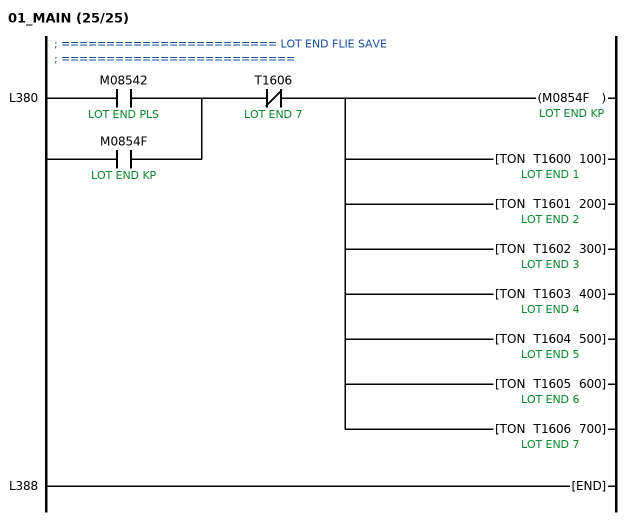
[picture p24: 01_MAIN rungs L380-L388]
// ======================== LOT END FLIE SAVE ==========================
; L380
LOAD      M08542	// LOT END PLS
OR        M0854F	// LOT END KP
AND NOT   T1606	// LOT END 7
OUT       M0854F	// LOT END KP
TON       T1600 100	// LOT END 1
TON       T1601 200	// LOT END 2
TON       T1602 300	// LOT END 3
TON       T1603 400	// LOT END 4
TON       T1604 500	// LOT END 5
TON       T1605 600	// LOT END 6
TON       T1606 700	// LOT END 7
; L388
END

PROGRAM 02_AUTO_RUN (task: ½ºÄµ ÇÁ·Î±×·¥)

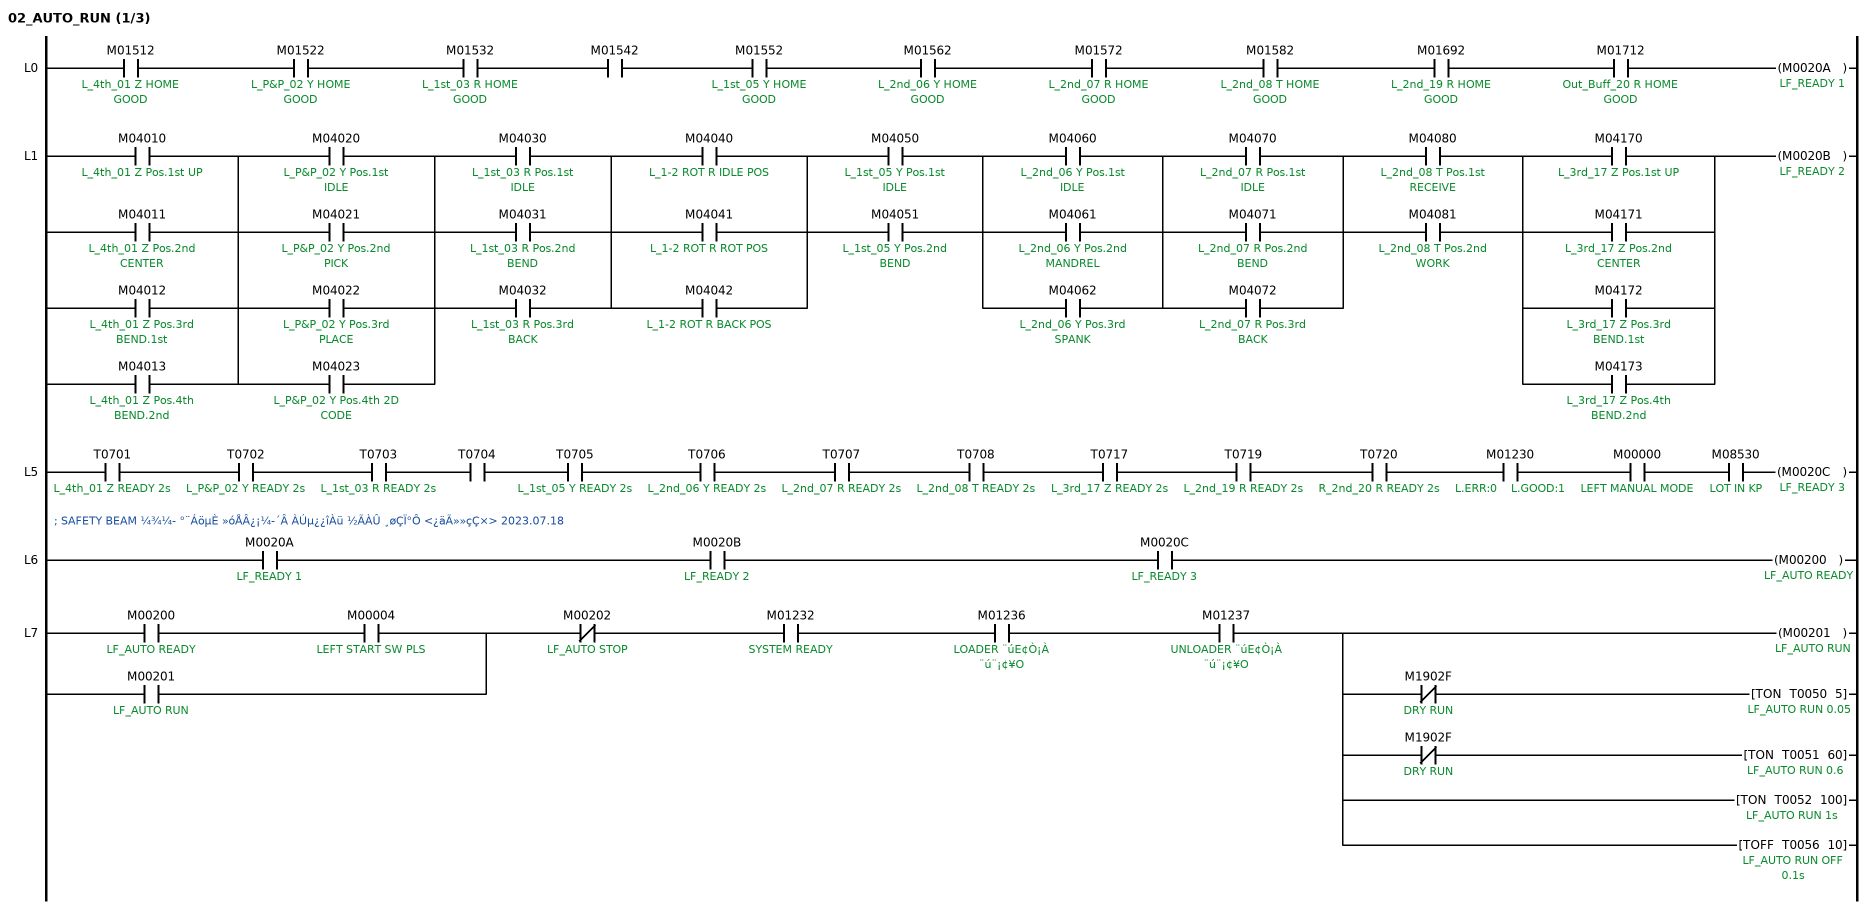
; L0
LOAD      M01512	// L_4th_01 Z HOME GOOD
AND       M01522	// L_P&P_02 Y HOME GOOD
AND       M01532	// L_1st_03 R HOME GOOD
AND       M01542
AND       M01552	// L_1st_05 Y HOME GOOD
AND       M01562	// L_2nd_06 Y HOME GOOD
AND       M01572	// L_2nd_07 R HOME GOOD
AND       M01582	// L_2nd_08 T HOME GOOD
AND       M01692	// L_2nd_19 R HOME GOOD
AND       M01712	// Out_Buff_20 R HOME GOOD
OUT       M0020A	// LF_READY 1
; L1
LOAD      M04010	// L_4th_01 Z Pos.1st UP
OR        M04011	// L_4th_01 Z Pos.2nd CENTER
OR        M04012	// L_4th_01 Z Pos.3rd BEND.1st
OR        M04013	// L_4th_01 Z Pos.4th BEND.2nd
LOAD      M04020	// L_P&P_02 Y Pos.1st IDLE
OR        M04021	// L_P&P_02 Y Pos.2nd PICK
OR        M04022	// L_P&P_02 Y Pos.3rd PLACE
OR        M04023	// L_P&P_02 Y Pos.4th 2D CODE
AND LOAD
LOAD      M04030	// L_1st_03 R Pos.1st IDLE
OR        M04031	// L_1st_03 R Pos.2nd BEND
OR        M04032	// L_1st_03 R Pos.3rd BACK
AND LOAD
LOAD      M04040	// L_1-2 ROT R IDLE POS
OR        M04041	// L_1-2 ROT R ROT POS
OR        M04042	// L_1-2 ROT R BACK POS
AND LOAD
LOAD      M04050	// L_1st_05 Y Pos.1st IDLE
OR        M04051	// L_1st_05 Y Pos.2nd BEND
AND LOAD
LOAD      M04060	// L_2nd_06 Y Pos.1st IDLE
OR        M04061	// L_2nd_06 Y Pos.2nd MANDREL
OR        M04062	// L_2nd_06 Y Pos.3rd SPANK
AND LOAD
LOAD      M04070	// L_2nd_07 R Pos.1st IDLE
OR        M04071	// L_2nd_07 R Pos.2nd BEND
OR        M04072	// L_2nd_07 R Pos.3rd BACK
AND LOAD
LOAD      M04080	// L_2nd_08 T Pos.1st RECEIVE
OR        M04081	// L_2nd_08 T Pos.2nd WORK
AND LOAD
LOAD      M04170	// L_3rd_17 Z Pos.1st UP
OR        M04171	// L_3rd_17 Z Pos.2nd CENTER
OR        M04172	// L_3rd_17 Z Pos.3rd BEND.1st
OR        M04173	// L_3rd_17 Z Pos.4th BEND.2nd
AND LOAD
OUT       M0020B	// LF_READY 2
; L5
LOAD      T0701	// L_4th_01 Z READY 2s
AND       T0702	// L_P&P_02 Y READY 2s
AND       T0703	// L_1st_03 R READY 2s
AND       T0704
AND       T0705	// L_1st_05 Y READY 2s
AND       T0706	// L_2nd_06 Y READY 2s
AND       T0707	// L_2nd_07 R READY 2s
AND       T0708	// L_2nd_08 T READY 2s
AND       T0717	// L_3rd_17 Z READY 2s
AND       T0719	// L_2nd_19 R READY 2s
AND       T0720	// R_2nd_20 R READY 2s
AND       M01230	// L.ERR:0    L.GOOD:1
AND       M00000	// LEFT MANUAL MODE
AND       M08530	// LOT IN KP
OUT       M0020C	// LF_READY 3
; L6
LOAD      M0020A	// LF_READY 1
AND       M0020B	// LF_READY 2
AND       M0020C	// LF_READY 3
OUT       M00200	// LF_AUTO READY
// output comment: SAFETY BEAM ¼¾¼­ °¨ÁöµÈ »óÅÂ¿¡¼­´Â ÀÚµ¿¿îÀü ½ÃÀÛ ¸øÇÏ°Ô <¿äÃ»»çÇ×> 2023.07.18
; L7
LOAD      M00200	// LF_AUTO READY
AND       M00004	// LEFT START SW PLS
OR        M00201	// LF_AUTO RUN
AND NOT   M00202	// LF_AUTO STOP
AND       M01232	// SYSTEM READY
AND       M01236	// LOADER ¨úE¢Ò¡À ¨ú¨¡¢¥O
AND       M01237	// UNLOADER ¨úE¢Ò¡À ¨ú¨¡¢¥O
OUT       M00201	// LF_AUTO RUN
MPUSH
AND NOT   M1902F	// DRY RUN
TON       T0050 5	// LF_AUTO RUN 0.05
MLOAD
AND NOT   M1902F	// DRY RUN
TON       T0051 60	// LF_AUTO RUN 0.6
MPOP
TON       T0052 100	// LF_AUTO RUN 1s
TOFF      T0056 10	// LF_AUTO RUN OFF 0.1s

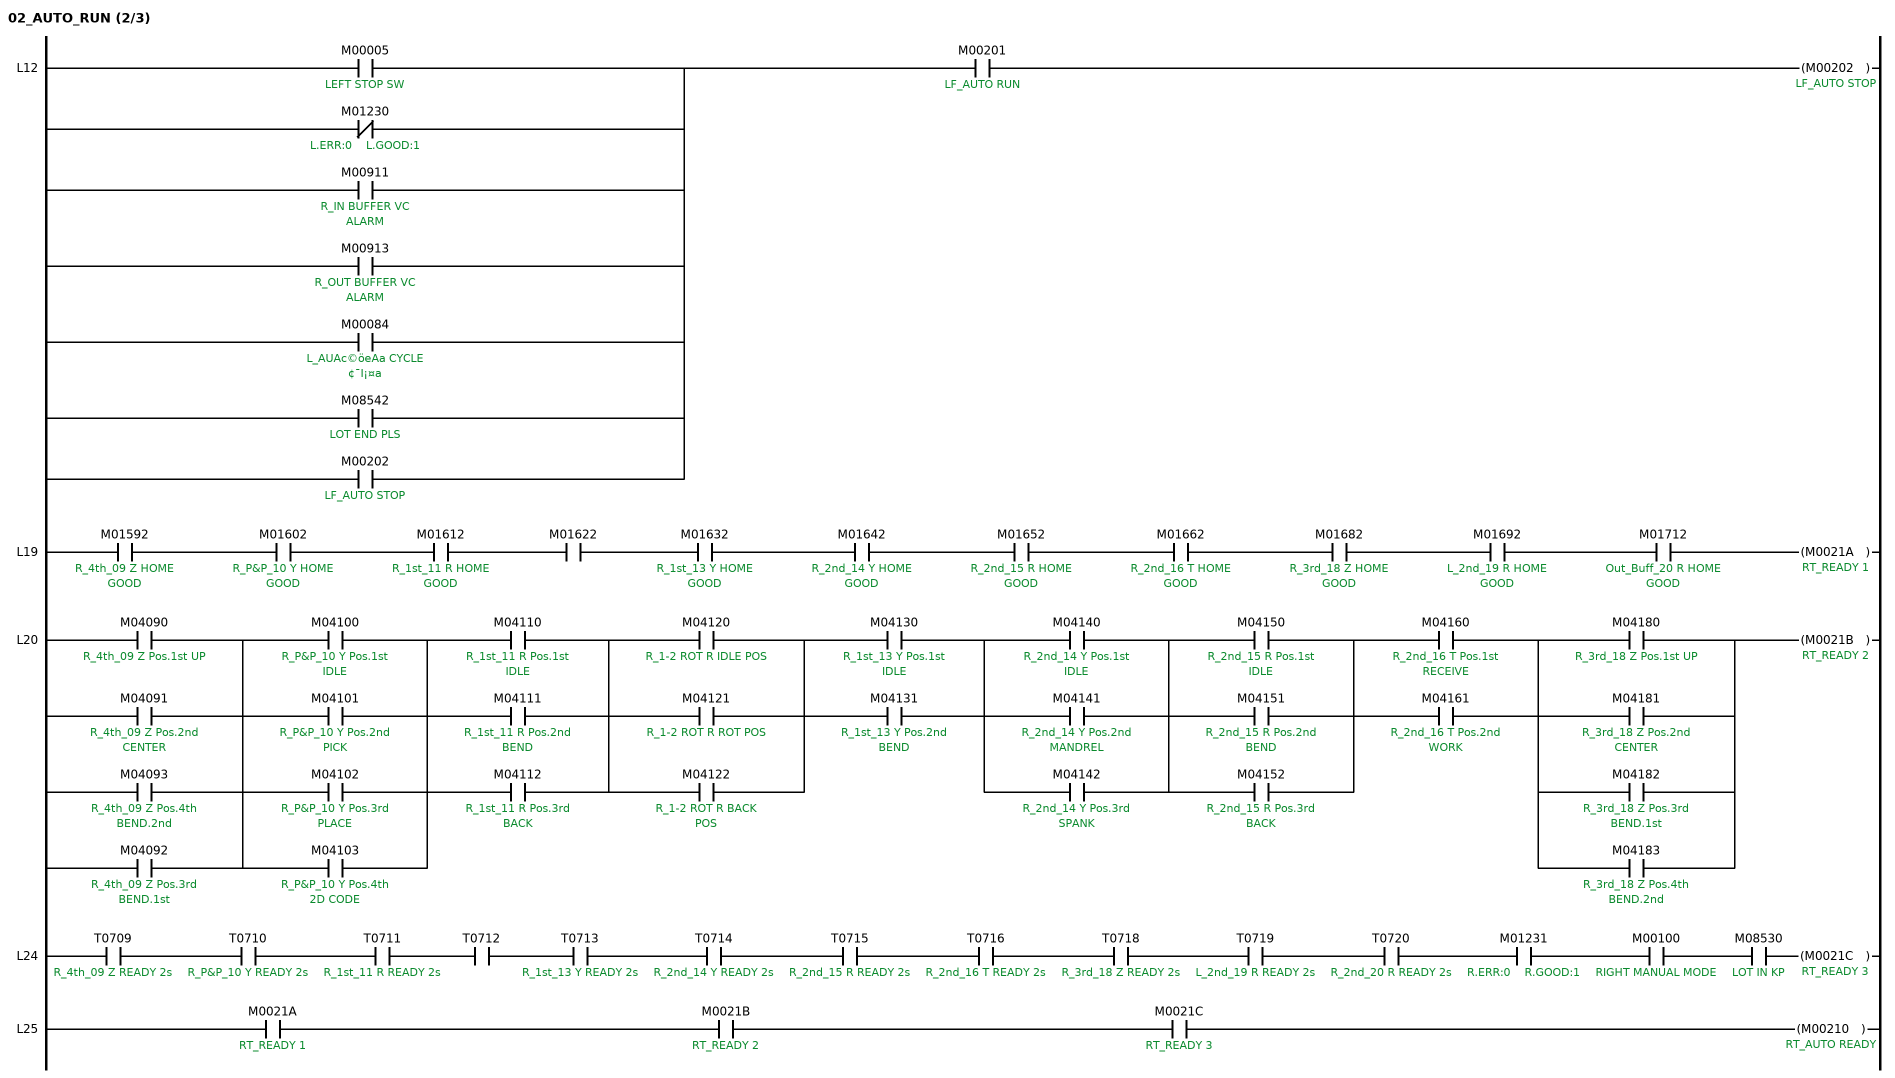
; L12
LOAD      M00005	// LEFT STOP SW
OR NOT    M01230	// L.ERR:0    L.GOOD:1
OR        M00911	// R_IN BUFFER VC ALARM
OR        M00913	// R_OUT BUFFER VC ALARM
OR        M00084	// L_AUAc©öeAa CYCLE ¢¯I¡¤a
OR        M08542	// LOT END PLS
OR        M00202	// LF_AUTO STOP
AND       M00201	// LF_AUTO RUN
OUT       M00202	// LF_AUTO STOP
; L19
LOAD      M01592	// R_4th_09 Z HOME GOOD
AND       M01602	// R_P&P_10 Y HOME GOOD
AND       M01612	// R_1st_11 R HOME GOOD
AND       M01622
AND       M01632	// R_1st_13 Y HOME GOOD
AND       M01642	// R_2nd_14 Y HOME GOOD
AND       M01652	// R_2nd_15 R HOME GOOD
AND       M01662	// R_2nd_16 T HOME GOOD
AND       M01682	// R_3rd_18 Z HOME GOOD
AND       M01692	// L_2nd_19 R HOME GOOD
AND       M01712	// Out_Buff_20 R HOME GOOD
OUT       M0021A	// RT_READY 1
; L20
LOAD      M04090	// R_4th_09 Z Pos.1st UP
OR        M04091	// R_4th_09 Z Pos.2nd CENTER
OR        M04093	// R_4th_09 Z Pos.4th BEND.2nd
OR        M04092	// R_4th_09 Z Pos.3rd BEND.1st
LOAD      M04100	// R_P&P_10 Y Pos.1st IDLE
OR        M04101	// R_P&P_10 Y Pos.2nd PICK
OR        M04102	// R_P&P_10 Y Pos.3rd PLACE
OR        M04103	// R_P&P_10 Y Pos.4th 2D CODE
AND LOAD
LOAD      M04110	// R_1st_11 R Pos.1st IDLE
OR        M04111	// R_1st_11 R Pos.2nd BEND
OR        M04112	// R_1st_11 R Pos.3rd BACK
AND LOAD
LOAD      M04120	// R_1-2 ROT R IDLE POS
OR        M04121	// R_1-2 ROT R ROT POS
OR        M04122	// R_1-2 ROT R BACK POS
AND LOAD
LOAD      M04130	// R_1st_13 Y Pos.1st IDLE
OR        M04131	// R_1st_13 Y Pos.2nd BEND
AND LOAD
LOAD      M04140	// R_2nd_14 Y Pos.1st IDLE
OR        M04141	// R_2nd_14 Y Pos.2nd MANDREL
OR        M04142	// R_2nd_14 Y Pos.3rd SPANK
AND LOAD
LOAD      M04150	// R_2nd_15 R Pos.1st IDLE
OR        M04151	// R_2nd_15 R Pos.2nd BEND
OR        M04152	// R_2nd_15 R Pos.3rd BACK
AND LOAD
LOAD      M04160	// R_2nd_16 T Pos.1st RECEIVE
OR        M04161	// R_2nd_16 T Pos.2nd WORK
AND LOAD
LOAD      M04180	// R_3rd_18 Z Pos.1st UP
OR        M04181	// R_3rd_18 Z Pos.2nd CENTER
OR        M04182	// R_3rd_18 Z Pos.3rd BEND.1st
OR        M04183	// R_3rd_18 Z Pos.4th BEND.2nd
AND LOAD
OUT       M0021B	// RT_READY 2
; L24
LOAD      T0709	// R_4th_09 Z READY 2s
AND       T0710	// R_P&P_10 Y READY 2s
AND       T0711	// R_1st_11 R READY 2s
AND       T0712
AND       T0713	// R_1st_13 Y READY 2s
AND       T0714	// R_2nd_14 Y READY 2s
AND       T0715	// R_2nd_15 R READY 2s
AND       T0716	// R_2nd_16 T READY 2s
AND       T0718	// R_3rd_18 Z READY 2s
AND       T0719	// L_2nd_19 R READY 2s
AND       T0720	// R_2nd_20 R READY 2s
AND       M01231	// R.ERR:0    R.GOOD:1
AND       M00100	// RIGHT MANUAL MODE
AND       M08530	// LOT IN KP
OUT       M0021C	// RT_READY 3
; L25
LOAD      M0021A	// RT_READY 1
AND       M0021B	// RT_READY 2
AND       M0021C	// RT_READY 3
OUT       M00210	// RT_AUTO READY

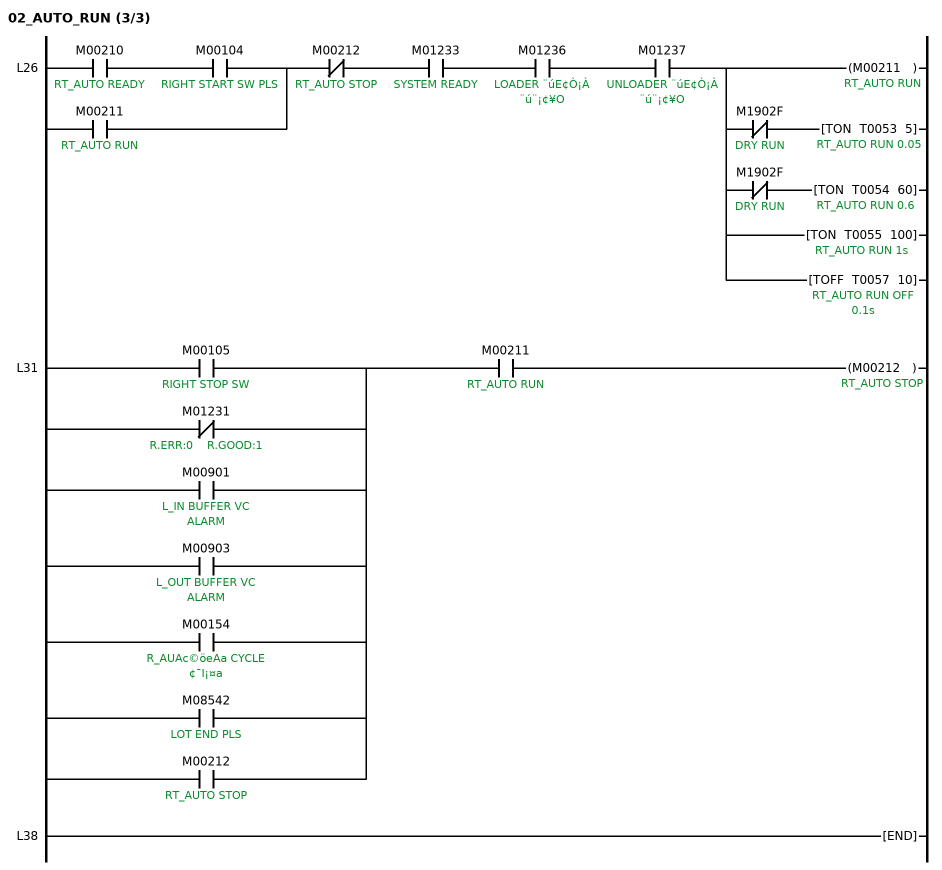
; L26
LOAD      M00210	// RT_AUTO READY
AND       M00104	// RIGHT START SW PLS
OR        M00211	// RT_AUTO RUN
AND NOT   M00212	// RT_AUTO STOP
AND       M01233	// SYSTEM READY
AND       M01236	// LOADER ¨úE¢Ò¡À ¨ú¨¡¢¥O
AND       M01237	// UNLOADER ¨úE¢Ò¡À ¨ú¨¡¢¥O
OUT       M00211	// RT_AUTO RUN
MPUSH
AND NOT   M1902F	// DRY RUN
TON       T0053 5	// RT_AUTO RUN 0.05
MLOAD
AND NOT   M1902F	// DRY RUN
TON       T0054 60	// RT_AUTO RUN 0.6
MPOP
TON       T0055 100	// RT_AUTO RUN 1s
TOFF      T0057 10	// RT_AUTO RUN OFF 0.1s
; L31
LOAD      M00105	// RIGHT STOP SW
OR NOT    M01231	// R.ERR:0    R.GOOD:1
OR        M00901	// L_IN BUFFER VC ALARM
OR        M00903	// L_OUT BUFFER VC ALARM
OR        M00154	// R_AUAc©öeAa CYCLE ¢¯I¡¤a
OR        M08542	// LOT END PLS
OR        M00212	// RT_AUTO STOP
AND       M00211	// RT_AUTO RUN
OUT       M00212	// RT_AUTO STOP
; L38
END

PROGRAM 03_COUNT (task: ½ºÄµ ÇÁ·Î±×·¥)

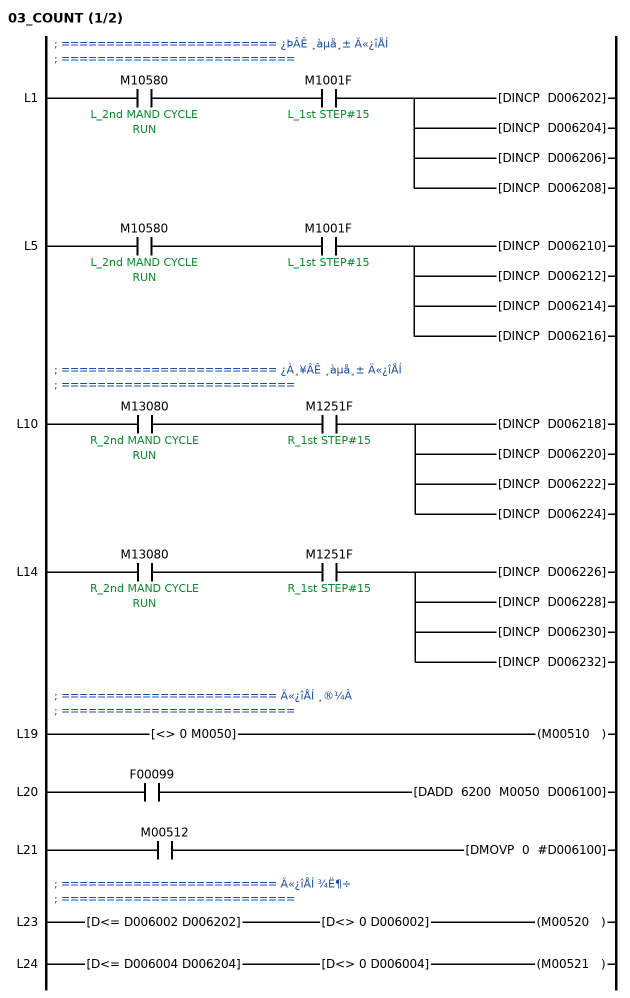
// ======================== ¿ÞÂÊ ¸àµå¸± Ä«¿îÅÍ ==========================
; L1
LOAD      M10580	// L_2nd MAND CYCLE RUN
AND       M1001F	// L_1st STEP#15
DINCP     D006202
DINCP     D006204
DINCP     D006206
DINCP     D006208
; L5
LOAD      M10580	// L_2nd MAND CYCLE RUN
AND       M1001F	// L_1st STEP#15
DINCP     D006210
DINCP     D006212
DINCP     D006214
DINCP     D006216
// ======================== ¿À¸¥ÂÊ ¸àµå¸± Ä«¿îÅÍ ==========================
; L10
LOAD      M13080	// R_2nd MAND CYCLE RUN
AND       M1251F	// R_1st STEP#15
DINCP     D006218
DINCP     D006220
DINCP     D006222
DINCP     D006224
; L14
LOAD      M13080	// R_2nd MAND CYCLE RUN
AND       M1251F	// R_1st STEP#15
DINCP     D006226
DINCP     D006228
DINCP     D006230
DINCP     D006232
// ======================== Ä«¿îÅÍ ¸®¼Â ==========================
; L19
LOAD<>    0 M0050
OUT       M00510
; L20
LOAD      F00099
DADD      6200 M0050 D006100
; L21
LOAD      M00512
DMOVP     0 #D006100
// ======================== Ä«¿îÅÍ ¾Ë¶÷ ==========================
; L23
LOADD<=   D006002 D006202
ANDD<>    0 D006002
OUT       M00520
; L24
LOADD<=   D006004 D006204
ANDD<>    0 D006004
OUT       M00521

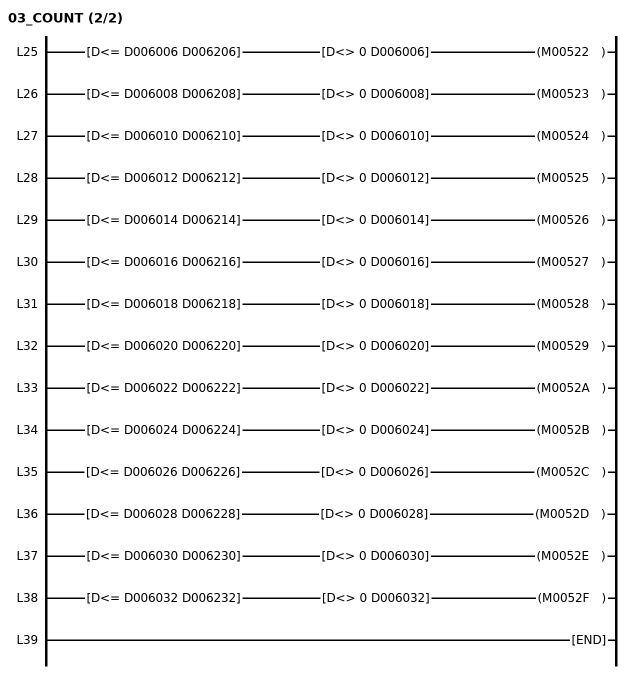
; L25
LOADD<=   D006006 D006206
ANDD<>    0 D006006
OUT       M00522
; L26
LOADD<=   D006008 D006208
ANDD<>    0 D006008
OUT       M00523
; L27
LOADD<=   D006010 D006210
ANDD<>    0 D006010
OUT       M00524
; L28
LOADD<=   D006012 D006212
ANDD<>    0 D006012
OUT       M00525
; L29
LOADD<=   D006014 D006214
ANDD<>    0 D006014
OUT       M00526
; L30
LOADD<=   D006016 D006216
ANDD<>    0 D006016
OUT       M00527
; L31
LOADD<=   D006018 D006218
ANDD<>    0 D006018
OUT       M00528
; L32
LOADD<=   D006020 D006220
ANDD<>    0 D006020
OUT       M00529
; L33
LOADD<=   D006022 D006222
ANDD<>    0 D006022
OUT       M0052A
; L34
LOADD<=   D006024 D006224
ANDD<>    0 D006024
OUT       M0052B
; L35
LOADD<=   D006026 D006226
ANDD<>    0 D006026
OUT       M0052C
; L36
LOADD<=   D006028 D006228
ANDD<>    0 D006028
OUT       M0052D
; L37
LOADD<=   D006030 D006230
ANDD<>    0 D006030
OUT       M0052E
; L38
LOADD<=   D006032 D006232
ANDD<>    0 D006032
OUT       M0052F
; L39
END

PROGRAM 04_VACUUM_FLOW (task: ½ºÄµ ÇÁ·Î±×·¥)

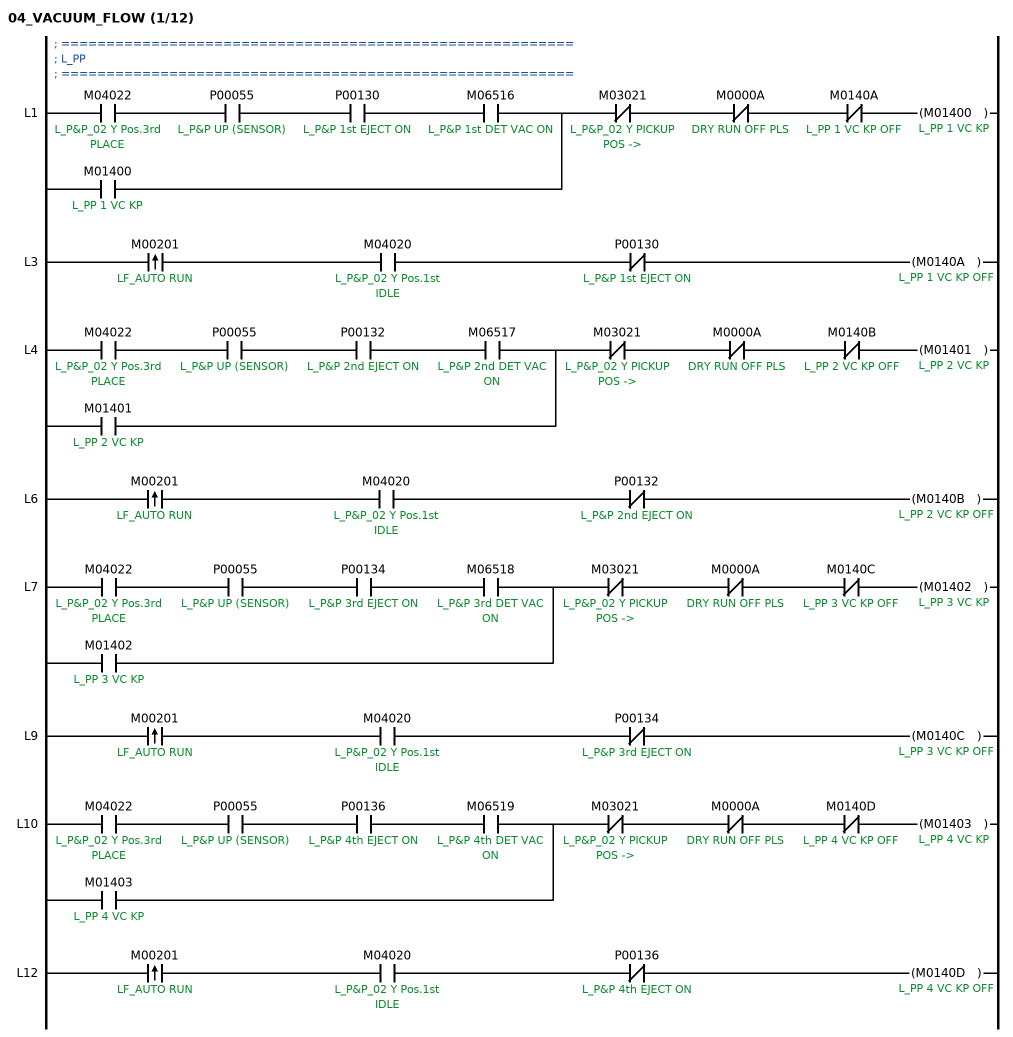
// =========================================================
// 
//       L_PP
// 
// =========================================================
; L1
LOAD      M04022	// L_P&P_02 Y Pos.3rd PLACE
AND       P00055	// L_P&P UP (SENSOR)
AND       P00130	// L_P&P 1st EJECT ON
AND       M06516	// L_P&P 1st DET VAC ON
OR        M01400	// L_PP 1 VC KP
AND NOT   M03021	// L_P&P_02 Y PICKUP POS ->
AND NOT   M0000A	// DRY RUN OFF PLS
AND NOT   M0140A	// L_PP 1 VC KP OFF
OUT       M01400	// L_PP 1 VC KP
; L3
LOADP     M00201	// LF_AUTO RUN
AND       M04020	// L_P&P_02 Y Pos.1st IDLE
AND NOT   P00130	// L_P&P 1st EJECT ON
OUT       M0140A	// L_PP 1 VC KP OFF
; L4
LOAD      M04022	// L_P&P_02 Y Pos.3rd PLACE
AND       P00055	// L_P&P UP (SENSOR)
AND       P00132	// L_P&P 2nd EJECT ON
AND       M06517	// L_P&P 2nd DET VAC ON
OR        M01401	// L_PP 2 VC KP
AND NOT   M03021	// L_P&P_02 Y PICKUP POS ->
AND NOT   M0000A	// DRY RUN OFF PLS
AND NOT   M0140B	// L_PP 2 VC KP OFF
OUT       M01401	// L_PP 2 VC KP
; L6
LOADP     M00201	// LF_AUTO RUN
AND       M04020	// L_P&P_02 Y Pos.1st IDLE
AND NOT   P00132	// L_P&P 2nd EJECT ON
OUT       M0140B	// L_PP 2 VC KP OFF
; L7
LOAD      M04022	// L_P&P_02 Y Pos.3rd PLACE
AND       P00055	// L_P&P UP (SENSOR)
AND       P00134	// L_P&P 3rd EJECT ON
AND       M06518	// L_P&P 3rd DET VAC ON
OR        M01402	// L_PP 3 VC KP
AND NOT   M03021	// L_P&P_02 Y PICKUP POS ->
AND NOT   M0000A	// DRY RUN OFF PLS
AND NOT   M0140C	// L_PP 3 VC KP OFF
OUT       M01402	// L_PP 3 VC KP
; L9
LOADP     M00201	// LF_AUTO RUN
AND       M04020	// L_P&P_02 Y Pos.1st IDLE
AND NOT   P00134	// L_P&P 3rd EJECT ON
OUT       M0140C	// L_PP 3 VC KP OFF
; L10
LOAD      M04022	// L_P&P_02 Y Pos.3rd PLACE
AND       P00055	// L_P&P UP (SENSOR)
AND       P00136	// L_P&P 4th EJECT ON
AND       M06519	// L_P&P 4th DET VAC ON
OR        M01403	// L_PP 4 VC KP
AND NOT   M03021	// L_P&P_02 Y PICKUP POS ->
AND NOT   M0000A	// DRY RUN OFF PLS
AND NOT   M0140D	// L_PP 4 VC KP OFF
OUT       M01403	// L_PP 4 VC KP
; L12
LOADP     M00201	// LF_AUTO RUN
AND       M04020	// L_P&P_02 Y Pos.1st IDLE
AND NOT   P00136	// L_P&P 4th EJECT ON
OUT       M0140D	// L_PP 4 VC KP OFF

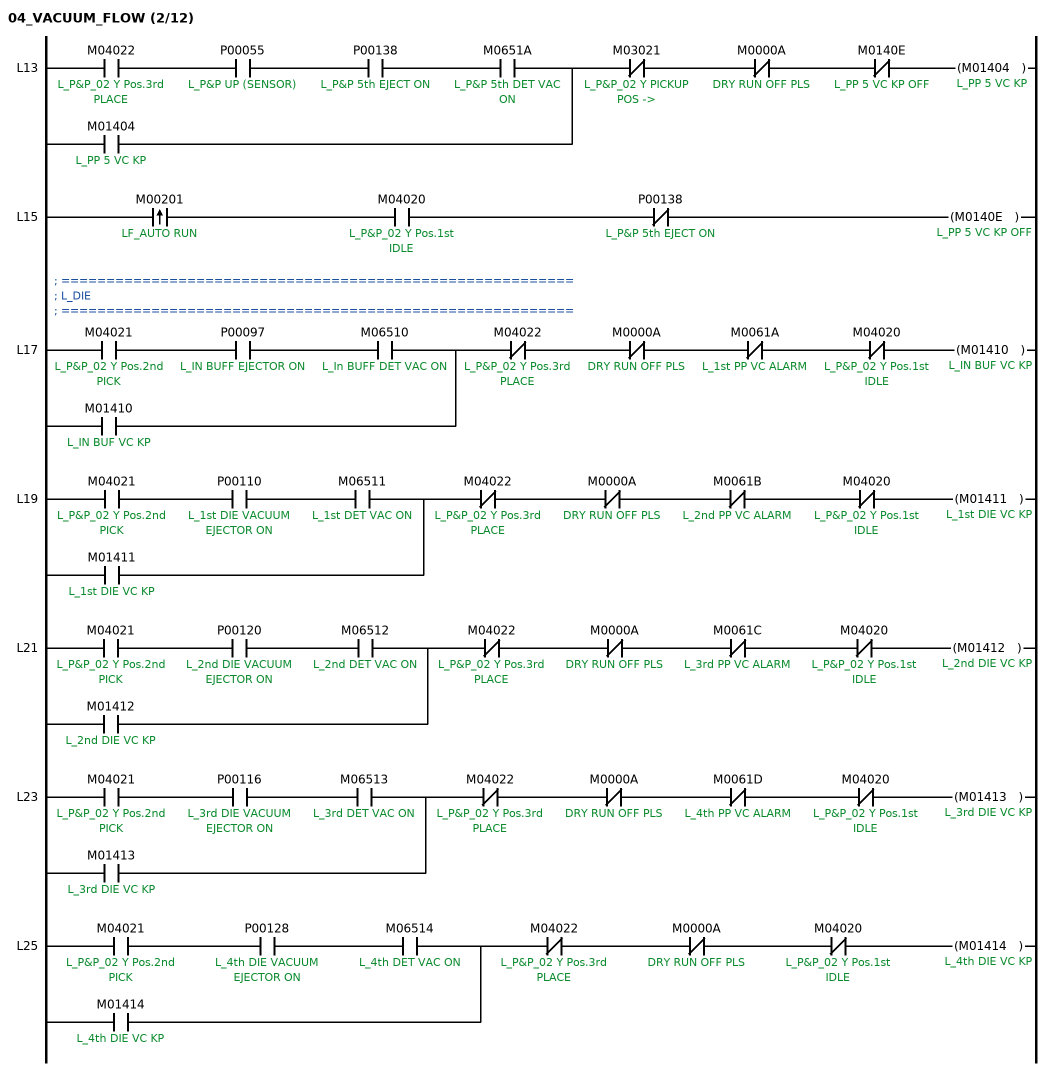
; L13
LOAD      M04022	// L_P&P_02 Y Pos.3rd PLACE
AND       P00055	// L_P&P UP (SENSOR)
AND       P00138	// L_P&P 5th EJECT ON
AND       M0651A	// L_P&P 5th DET VAC ON
OR        M01404	// L_PP 5 VC KP
AND NOT   M03021	// L_P&P_02 Y PICKUP POS ->
AND NOT   M0000A	// DRY RUN OFF PLS
AND NOT   M0140E	// L_PP 5 VC KP OFF
OUT       M01404	// L_PP 5 VC KP
; L15
LOADP     M00201	// LF_AUTO RUN
AND       M04020	// L_P&P_02 Y Pos.1st IDLE
AND NOT   P00138	// L_P&P 5th EJECT ON
OUT       M0140E	// L_PP 5 VC KP OFF
// =========================================================
// 
//       L_DIE
// 
// =========================================================
; L17
LOAD      M04021	// L_P&P_02 Y Pos.2nd PICK
AND       P00097	// L_IN BUFF EJECTOR ON
AND       M06510	// L_In BUFF DET VAC ON
OR        M01410	// L_IN BUF VC KP
AND NOT   M04022	// L_P&P_02 Y Pos.3rd PLACE
AND NOT   M0000A	// DRY RUN OFF PLS
AND NOT   M0061A	// L_1st PP VC ALARM
AND NOT   M04020	// L_P&P_02 Y Pos.1st IDLE
OUT       M01410	// L_IN BUF VC KP
; L19
LOAD      M04021	// L_P&P_02 Y Pos.2nd PICK
AND       P00110	// L_1st DIE VACUUM EJECTOR ON
AND       M06511	// L_1st DET VAC ON
OR        M01411	// L_1st DIE VC KP
AND NOT   M04022	// L_P&P_02 Y Pos.3rd PLACE
AND NOT   M0000A	// DRY RUN OFF PLS
AND NOT   M0061B	// L_2nd PP VC ALARM
AND NOT   M04020	// L_P&P_02 Y Pos.1st IDLE
OUT       M01411	// L_1st DIE VC KP
; L21
LOAD      M04021	// L_P&P_02 Y Pos.2nd PICK
AND       P00120	// L_2nd DIE VACUUM EJECTOR ON
AND       M06512	// L_2nd DET VAC ON
OR        M01412	// L_2nd DIE VC KP
AND NOT   M04022	// L_P&P_02 Y Pos.3rd PLACE
AND NOT   M0000A	// DRY RUN OFF PLS
AND NOT   M0061C	// L_3rd PP VC ALARM
AND NOT   M04020	// L_P&P_02 Y Pos.1st IDLE
OUT       M01412	// L_2nd DIE VC KP
; L23
LOAD      M04021	// L_P&P_02 Y Pos.2nd PICK
AND       P00116	// L_3rd DIE VACUUM EJECTOR ON
AND       M06513	// L_3rd DET VAC ON
OR        M01413	// L_3rd DIE VC KP
AND NOT   M04022	// L_P&P_02 Y Pos.3rd PLACE
AND NOT   M0000A	// DRY RUN OFF PLS
AND NOT   M0061D	// L_4th PP VC ALARM
AND NOT   M04020	// L_P&P_02 Y Pos.1st IDLE
OUT       M01413	// L_3rd DIE VC KP
; L25
LOAD      M04021	// L_P&P_02 Y Pos.2nd PICK
AND       P00128	// L_4th DIE VACUUM EJECTOR ON
AND       M06514	// L_4th DET VAC ON
OR        M01414	// L_4th DIE VC KP
AND NOT   M04022	// L_P&P_02 Y Pos.3rd PLACE
AND NOT   M0000A	// DRY RUN OFF PLS
AND NOT   M04020	// L_P&P_02 Y Pos.1st IDLE
OUT       M01414	// L_4th DIE VC KP

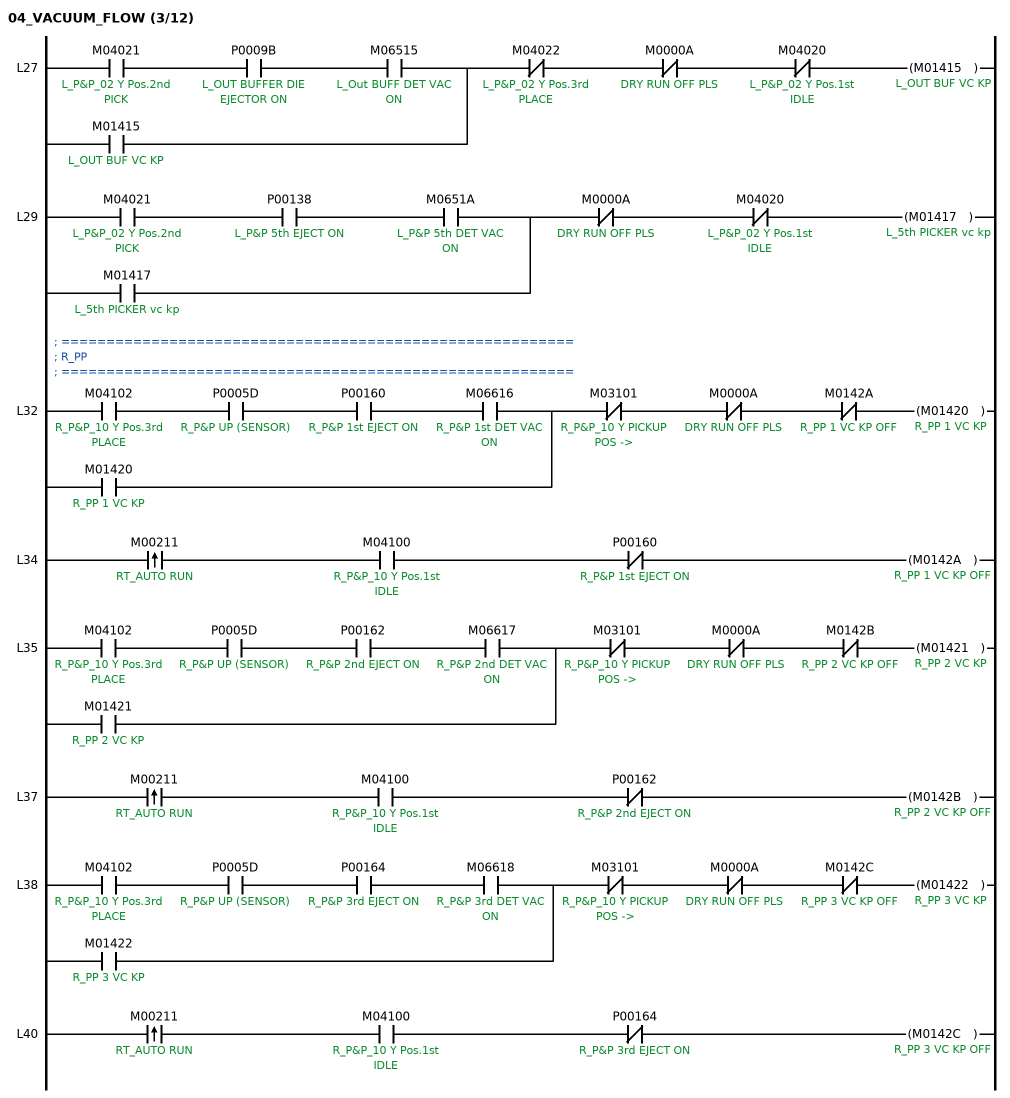
; L27
LOAD      M04021	// L_P&P_02 Y Pos.2nd PICK
AND       P0009B	// L_OUT BUFFER DIE EJECTOR ON
AND       M06515	// L_Out BUFF DET VAC ON
OR        M01415	// L_OUT BUF VC KP
AND NOT   M04022	// L_P&P_02 Y Pos.3rd PLACE
AND NOT   M0000A	// DRY RUN OFF PLS
AND NOT   M04020	// L_P&P_02 Y Pos.1st IDLE
OUT       M01415	// L_OUT BUF VC KP
; L29
LOAD      M04021	// L_P&P_02 Y Pos.2nd PICK
AND       P00138	// L_P&P 5th EJECT ON
AND       M0651A	// L_P&P 5th DET VAC ON
OR        M01417	// L_5th PICKER vc kp
AND NOT   M0000A	// DRY RUN OFF PLS
AND NOT   M04020	// L_P&P_02 Y Pos.1st IDLE
OUT       M01417	// L_5th PICKER vc kp
// =========================================================
// 
//       R_PP
// 
// =========================================================
; L32
LOAD      M04102	// R_P&P_10 Y Pos.3rd PLACE
AND       P0005D	// R_P&P UP (SENSOR)
AND       P00160	// R_P&P 1st EJECT ON
AND       M06616	// R_P&P 1st DET VAC ON
OR        M01420	// R_PP 1 VC KP
AND NOT   M03101	// R_P&P_10 Y PICKUP POS ->
AND NOT   M0000A	// DRY RUN OFF PLS
AND NOT   M0142A	// R_PP 1 VC KP OFF
OUT       M01420	// R_PP 1 VC KP
; L34
LOADP     M00211	// RT_AUTO RUN
AND       M04100	// R_P&P_10 Y Pos.1st IDLE
AND NOT   P00160	// R_P&P 1st EJECT ON
OUT       M0142A	// R_PP 1 VC KP OFF
; L35
LOAD      M04102	// R_P&P_10 Y Pos.3rd PLACE
AND       P0005D	// R_P&P UP (SENSOR)
AND       P00162	// R_P&P 2nd EJECT ON
AND       M06617	// R_P&P 2nd DET VAC ON
OR        M01421	// R_PP 2 VC KP
AND NOT   M03101	// R_P&P_10 Y PICKUP POS ->
AND NOT   M0000A	// DRY RUN OFF PLS
AND NOT   M0142B	// R_PP 2 VC KP OFF
OUT       M01421	// R_PP 2 VC KP
; L37
LOADP     M00211	// RT_AUTO RUN
AND       M04100	// R_P&P_10 Y Pos.1st IDLE
AND NOT   P00162	// R_P&P 2nd EJECT ON
OUT       M0142B	// R_PP 2 VC KP OFF
; L38
LOAD      M04102	// R_P&P_10 Y Pos.3rd PLACE
AND       P0005D	// R_P&P UP (SENSOR)
AND       P00164	// R_P&P 3rd EJECT ON
AND       M06618	// R_P&P 3rd DET VAC ON
OR        M01422	// R_PP 3 VC KP
AND NOT   M03101	// R_P&P_10 Y PICKUP POS ->
AND NOT   M0000A	// DRY RUN OFF PLS
AND NOT   M0142C	// R_PP 3 VC KP OFF
OUT       M01422	// R_PP 3 VC KP
; L40
LOADP     M00211	// RT_AUTO RUN
AND       M04100	// R_P&P_10 Y Pos.1st IDLE
AND NOT   P00164	// R_P&P 3rd EJECT ON
OUT       M0142C	// R_PP 3 VC KP OFF

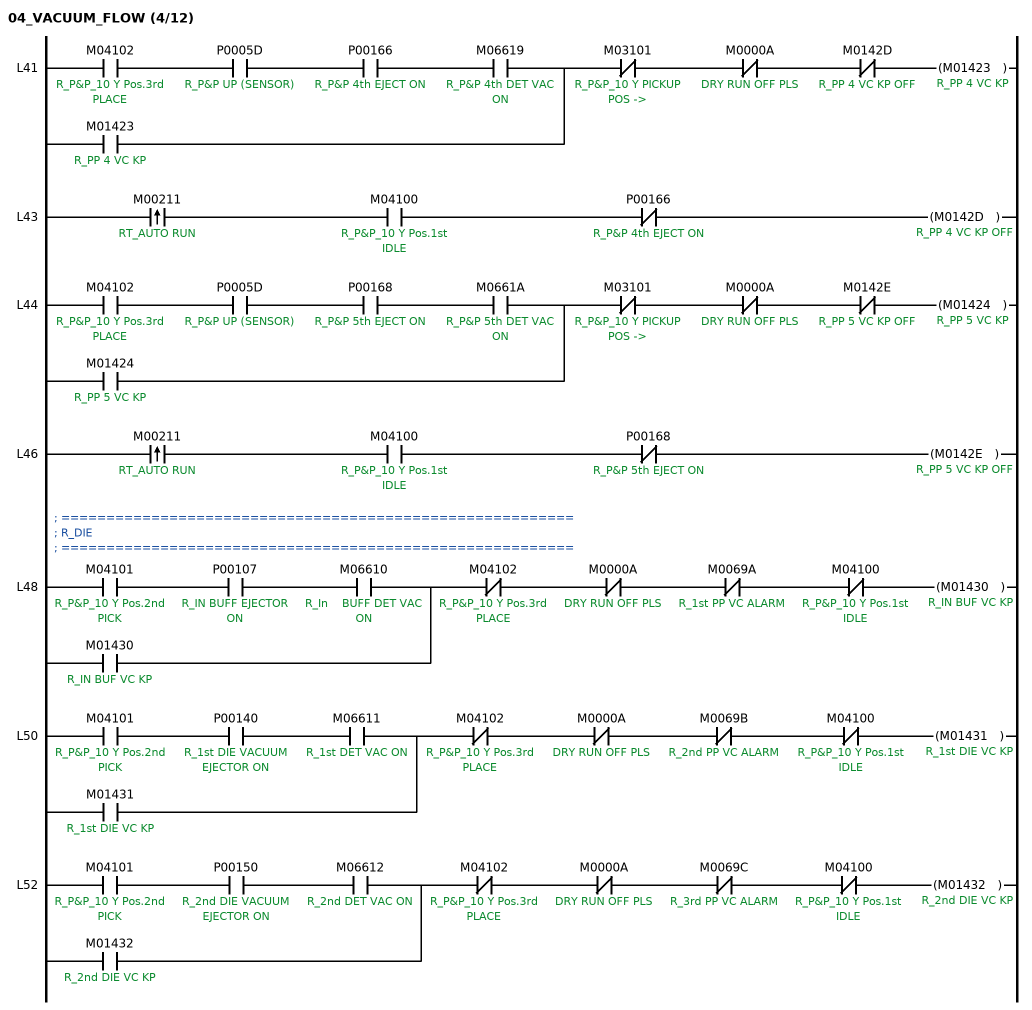
; L41
LOAD      M04102	// R_P&P_10 Y Pos.3rd PLACE
AND       P0005D	// R_P&P UP (SENSOR)
AND       P00166	// R_P&P 4th EJECT ON
AND       M06619	// R_P&P 4th DET VAC ON
OR        M01423	// R_PP 4 VC KP
AND NOT   M03101	// R_P&P_10 Y PICKUP POS ->
AND NOT   M0000A	// DRY RUN OFF PLS
AND NOT   M0142D	// R_PP 4 VC KP OFF
OUT       M01423	// R_PP 4 VC KP
; L43
LOADP     M00211	// RT_AUTO RUN
AND       M04100	// R_P&P_10 Y Pos.1st IDLE
AND NOT   P00166	// R_P&P 4th EJECT ON
OUT       M0142D	// R_PP 4 VC KP OFF
; L44
LOAD      M04102	// R_P&P_10 Y Pos.3rd PLACE
AND       P0005D	// R_P&P UP (SENSOR)
AND       P00168	// R_P&P 5th EJECT ON
AND       M0661A	// R_P&P 5th DET VAC ON
OR        M01424	// R_PP 5 VC KP
AND NOT   M03101	// R_P&P_10 Y PICKUP POS ->
AND NOT   M0000A	// DRY RUN OFF PLS
AND NOT   M0142E	// R_PP 5 VC KP OFF
OUT       M01424	// R_PP 5 VC KP
; L46
LOADP     M00211	// RT_AUTO RUN
AND       M04100	// R_P&P_10 Y Pos.1st IDLE
AND NOT   P00168	// R_P&P 5th EJECT ON
OUT       M0142E	// R_PP 5 VC KP OFF
// =========================================================
// 
//       R_DIE
// 
// =========================================================
; L48
LOAD      M04101	// R_P&P_10 Y Pos.2nd PICK
AND       P00107	// R_IN BUFF EJECTOR ON
AND       M06610	// R_In    BUFF DET VAC ON
OR        M01430	// R_IN BUF VC KP
AND NOT   M04102	// R_P&P_10 Y Pos.3rd PLACE
AND NOT   M0000A	// DRY RUN OFF PLS
AND NOT   M0069A	// R_1st PP VC ALARM
AND NOT   M04100	// R_P&P_10 Y Pos.1st IDLE
OUT       M01430	// R_IN BUF VC KP
; L50
LOAD      M04101	// R_P&P_10 Y Pos.2nd PICK
AND       P00140	// R_1st DIE VACUUM EJECTOR ON
AND       M06611	// R_1st DET VAC ON
OR        M01431	// R_1st DIE VC KP
AND NOT   M04102	// R_P&P_10 Y Pos.3rd PLACE
AND NOT   M0000A	// DRY RUN OFF PLS
AND NOT   M0069B	// R_2nd PP VC ALARM
AND NOT   M04100	// R_P&P_10 Y Pos.1st IDLE
OUT       M01431	// R_1st DIE VC KP
; L52
LOAD      M04101	// R_P&P_10 Y Pos.2nd PICK
AND       P00150	// R_2nd DIE VACUUM EJECTOR ON
AND       M06612	// R_2nd DET VAC ON
OR        M01432	// R_2nd DIE VC KP
AND NOT   M04102	// R_P&P_10 Y Pos.3rd PLACE
AND NOT   M0000A	// DRY RUN OFF PLS
AND NOT   M0069C	// R_3rd PP VC ALARM
AND NOT   M04100	// R_P&P_10 Y Pos.1st IDLE
OUT       M01432	// R_2nd DIE VC KP

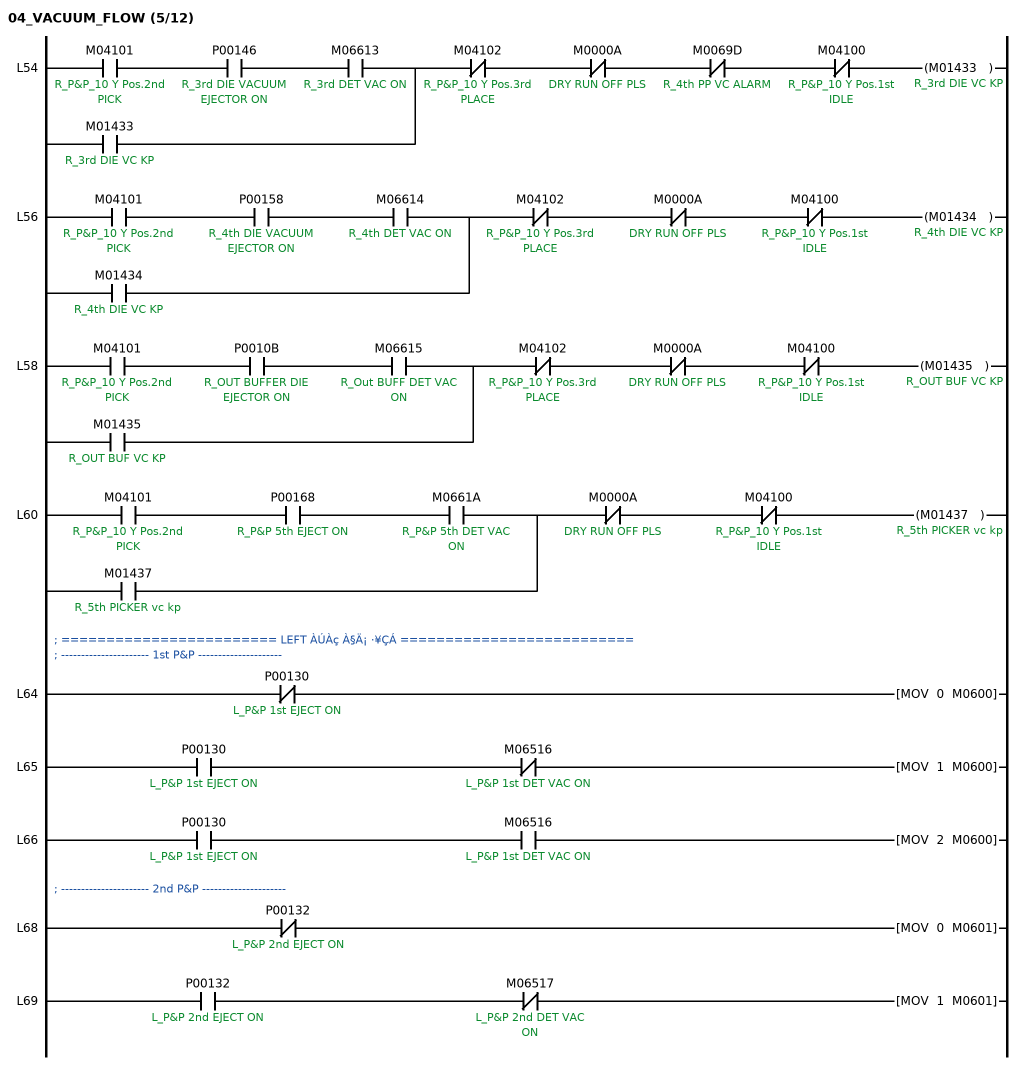
; L54
LOAD      M04101	// R_P&P_10 Y Pos.2nd PICK
AND       P00146	// R_3rd DIE VACUUM EJECTOR ON
AND       M06613	// R_3rd DET VAC ON
OR        M01433	// R_3rd DIE VC KP
AND NOT   M04102	// R_P&P_10 Y Pos.3rd PLACE
AND NOT   M0000A	// DRY RUN OFF PLS
AND NOT   M0069D	// R_4th PP VC ALARM
AND NOT   M04100	// R_P&P_10 Y Pos.1st IDLE
OUT       M01433	// R_3rd DIE VC KP
; L56
LOAD      M04101	// R_P&P_10 Y Pos.2nd PICK
AND       P00158	// R_4th DIE VACUUM EJECTOR ON
AND       M06614	// R_4th DET VAC ON
OR        M01434	// R_4th DIE VC KP
AND NOT   M04102	// R_P&P_10 Y Pos.3rd PLACE
AND NOT   M0000A	// DRY RUN OFF PLS
AND NOT   M04100	// R_P&P_10 Y Pos.1st IDLE
OUT       M01434	// R_4th DIE VC KP
; L58
LOAD      M04101	// R_P&P_10 Y Pos.2nd PICK
AND       P0010B	// R_OUT BUFFER DIE EJECTOR ON
AND       M06615	// R_Out BUFF DET VAC ON
OR        M01435	// R_OUT BUF VC KP
AND NOT   M04102	// R_P&P_10 Y Pos.3rd PLACE
AND NOT   M0000A	// DRY RUN OFF PLS
AND NOT   M04100	// R_P&P_10 Y Pos.1st IDLE
OUT       M01435	// R_OUT BUF VC KP
; L60
LOAD      M04101	// R_P&P_10 Y Pos.2nd PICK
AND       P00168	// R_P&P 5th EJECT ON
AND       M0661A	// R_P&P 5th DET VAC ON
OR        M01437	// R_5th PICKER vc kp
AND NOT   M0000A	// DRY RUN OFF PLS
AND NOT   M04100	// R_P&P_10 Y Pos.1st IDLE
OUT       M01437	// R_5th PICKER vc kp
// ======================== LEFT ÀÚÀç À§Ä¡ ·¥ÇÁ ==========================
// ---------------------- 1st P&P ---------------------
; L64
LOAD NOT  P00130	// L_P&P 1st EJECT ON
MOV       0 M0600
; L65
LOAD      P00130	// L_P&P 1st EJECT ON
AND NOT   M06516	// L_P&P 1st DET VAC ON
MOV       1 M0600
; L66
LOAD      P00130	// L_P&P 1st EJECT ON
AND       M06516	// L_P&P 1st DET VAC ON
MOV       2 M0600
// ---------------------- 2nd P&P ---------------------
; L68
LOAD NOT  P00132	// L_P&P 2nd EJECT ON
MOV       0 M0601
; L69
LOAD      P00132	// L_P&P 2nd EJECT ON
AND NOT   M06517	// L_P&P 2nd DET VAC ON
MOV       1 M0601

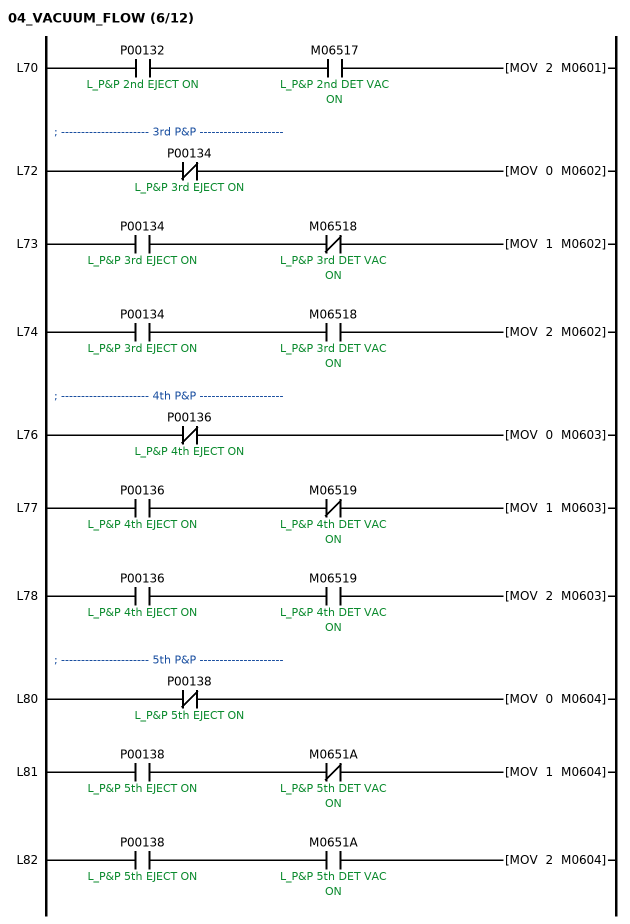
; L70
LOAD      P00132	// L_P&P 2nd EJECT ON
AND       M06517	// L_P&P 2nd DET VAC ON
MOV       2 M0601
// ---------------------- 3rd P&P ---------------------
; L72
LOAD NOT  P00134	// L_P&P 3rd EJECT ON
MOV       0 M0602
; L73
LOAD      P00134	// L_P&P 3rd EJECT ON
AND NOT   M06518	// L_P&P 3rd DET VAC ON
MOV       1 M0602
; L74
LOAD      P00134	// L_P&P 3rd EJECT ON
AND       M06518	// L_P&P 3rd DET VAC ON
MOV       2 M0602
// ---------------------- 4th P&P ---------------------
; L76
LOAD NOT  P00136	// L_P&P 4th EJECT ON
MOV       0 M0603
; L77
LOAD      P00136	// L_P&P 4th EJECT ON
AND NOT   M06519	// L_P&P 4th DET VAC ON
MOV       1 M0603
; L78
LOAD      P00136	// L_P&P 4th EJECT ON
AND       M06519	// L_P&P 4th DET VAC ON
MOV       2 M0603
// ---------------------- 5th P&P ---------------------
; L80
LOAD NOT  P00138	// L_P&P 5th EJECT ON
MOV       0 M0604
; L81
LOAD      P00138	// L_P&P 5th EJECT ON
AND NOT   M0651A	// L_P&P 5th DET VAC ON
MOV       1 M0604
; L82
LOAD      P00138	// L_P&P 5th EJECT ON
AND       M0651A	// L_P&P 5th DET VAC ON
MOV       2 M0604

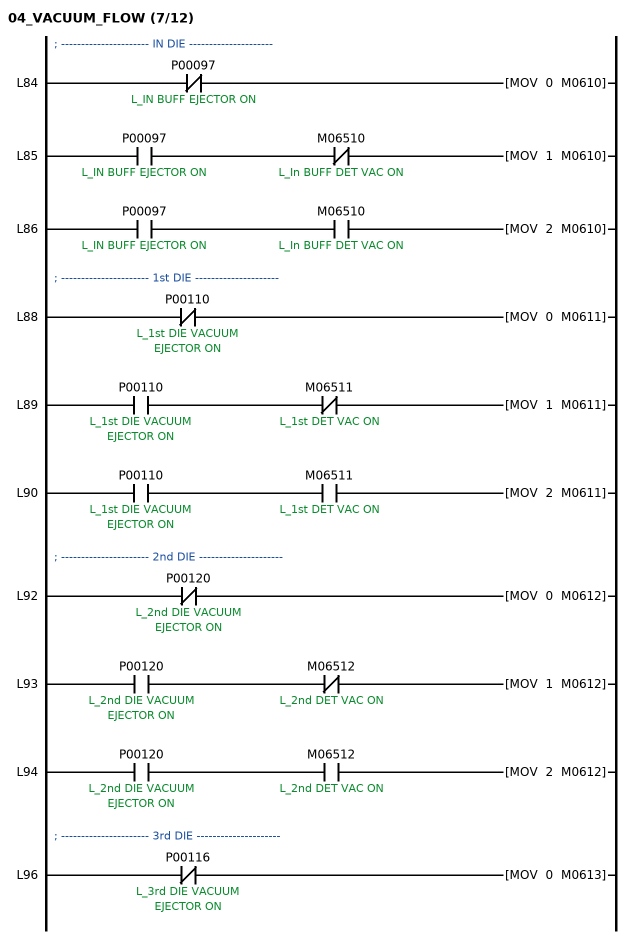
// ---------------------- IN DIE ---------------------
; L84
LOAD NOT  P00097	// L_IN BUFF EJECTOR ON
MOV       0 M0610
; L85
LOAD      P00097	// L_IN BUFF EJECTOR ON
AND NOT   M06510	// L_In BUFF DET VAC ON
MOV       1 M0610
; L86
LOAD      P00097	// L_IN BUFF EJECTOR ON
AND       M06510	// L_In BUFF DET VAC ON
MOV       2 M0610
// ---------------------- 1st DIE ---------------------
; L88
LOAD NOT  P00110	// L_1st DIE VACUUM EJECTOR ON
MOV       0 M0611
; L89
LOAD      P00110	// L_1st DIE VACUUM EJECTOR ON
AND NOT   M06511	// L_1st DET VAC ON
MOV       1 M0611
; L90
LOAD      P00110	// L_1st DIE VACUUM EJECTOR ON
AND       M06511	// L_1st DET VAC ON
MOV       2 M0611
// ---------------------- 2nd DIE ---------------------
; L92
LOAD NOT  P00120	// L_2nd DIE VACUUM EJECTOR ON
MOV       0 M0612
; L93
LOAD      P00120	// L_2nd DIE VACUUM EJECTOR ON
AND NOT   M06512	// L_2nd DET VAC ON
MOV       1 M0612
; L94
LOAD      P00120	// L_2nd DIE VACUUM EJECTOR ON
AND       M06512	// L_2nd DET VAC ON
MOV       2 M0612
// ---------------------- 3rd DIE ---------------------
; L96
LOAD NOT  P00116	// L_3rd DIE VACUUM EJECTOR ON
MOV       0 M0613

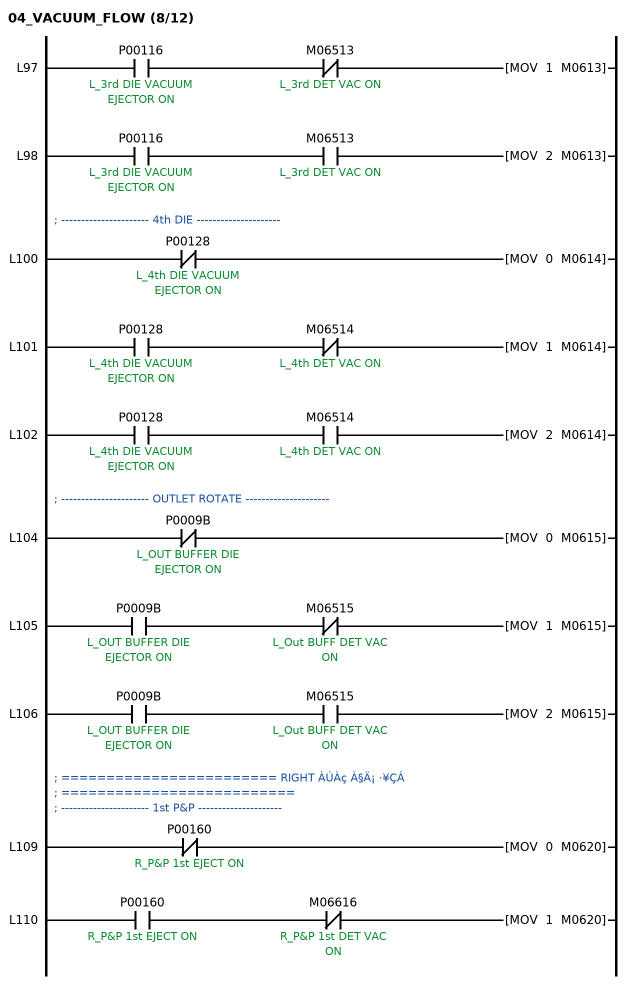
; L97
LOAD      P00116	// L_3rd DIE VACUUM EJECTOR ON
AND NOT   M06513	// L_3rd DET VAC ON
MOV       1 M0613
; L98
LOAD      P00116	// L_3rd DIE VACUUM EJECTOR ON
AND       M06513	// L_3rd DET VAC ON
MOV       2 M0613
// ---------------------- 4th DIE ---------------------
; L100
LOAD NOT  P00128	// L_4th DIE VACUUM EJECTOR ON
MOV       0 M0614
; L101
LOAD      P00128	// L_4th DIE VACUUM EJECTOR ON
AND NOT   M06514	// L_4th DET VAC ON
MOV       1 M0614
; L102
LOAD      P00128	// L_4th DIE VACUUM EJECTOR ON
AND       M06514	// L_4th DET VAC ON
MOV       2 M0614
// ---------------------- OUTLET ROTATE ---------------------
; L104
LOAD NOT  P0009B	// L_OUT BUFFER DIE EJECTOR ON
MOV       0 M0615
; L105
LOAD      P0009B	// L_OUT BUFFER DIE EJECTOR ON
AND NOT   M06515	// L_Out BUFF DET VAC ON
MOV       1 M0615
; L106
LOAD      P0009B	// L_OUT BUFFER DIE EJECTOR ON
AND       M06515	// L_Out BUFF DET VAC ON
MOV       2 M0615
// ======================== RIGHT ÀÚÀç À§Ä¡ ·¥ÇÁ ==========================
// ---------------------- 1st P&P ---------------------
; L109
LOAD NOT  P00160	// R_P&P 1st EJECT ON
MOV       0 M0620
; L110
LOAD      P00160	// R_P&P 1st EJECT ON
AND NOT   M06616	// R_P&P 1st DET VAC ON
MOV       1 M0620

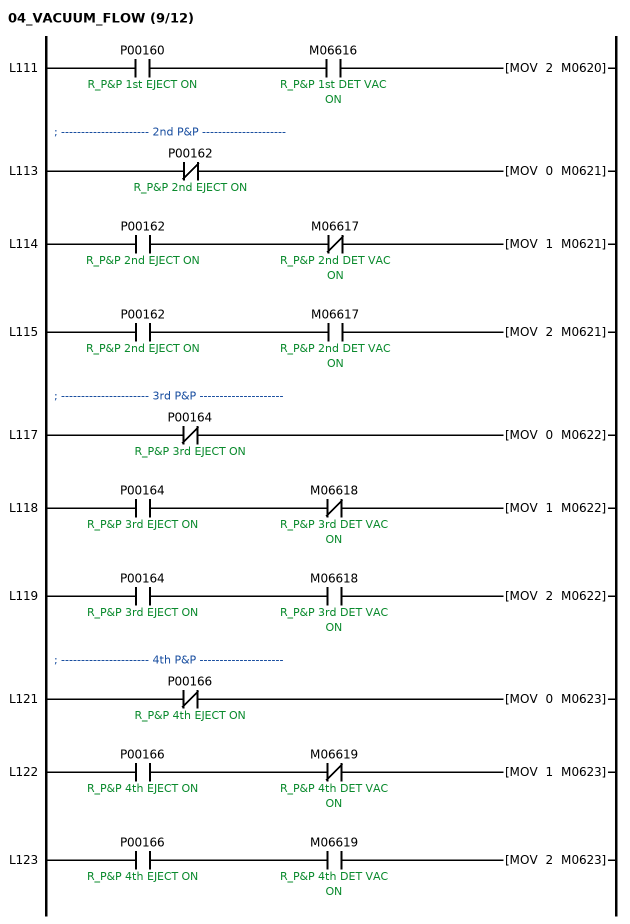
; L111
LOAD      P00160	// R_P&P 1st EJECT ON
AND       M06616	// R_P&P 1st DET VAC ON
MOV       2 M0620
// ---------------------- 2nd P&P ---------------------
; L113
LOAD NOT  P00162	// R_P&P 2nd EJECT ON
MOV       0 M0621
; L114
LOAD      P00162	// R_P&P 2nd EJECT ON
AND NOT   M06617	// R_P&P 2nd DET VAC ON
MOV       1 M0621
; L115
LOAD      P00162	// R_P&P 2nd EJECT ON
AND       M06617	// R_P&P 2nd DET VAC ON
MOV       2 M0621
// ---------------------- 3rd P&P ---------------------
; L117
LOAD NOT  P00164	// R_P&P 3rd EJECT ON
MOV       0 M0622
; L118
LOAD      P00164	// R_P&P 3rd EJECT ON
AND NOT   M06618	// R_P&P 3rd DET VAC ON
MOV       1 M0622
; L119
LOAD      P00164	// R_P&P 3rd EJECT ON
AND       M06618	// R_P&P 3rd DET VAC ON
MOV       2 M0622
// ---------------------- 4th P&P ---------------------
; L121
LOAD NOT  P00166	// R_P&P 4th EJECT ON
MOV       0 M0623
; L122
LOAD      P00166	// R_P&P 4th EJECT ON
AND NOT   M06619	// R_P&P 4th DET VAC ON
MOV       1 M0623
; L123
LOAD      P00166	// R_P&P 4th EJECT ON
AND       M06619	// R_P&P 4th DET VAC ON
MOV       2 M0623

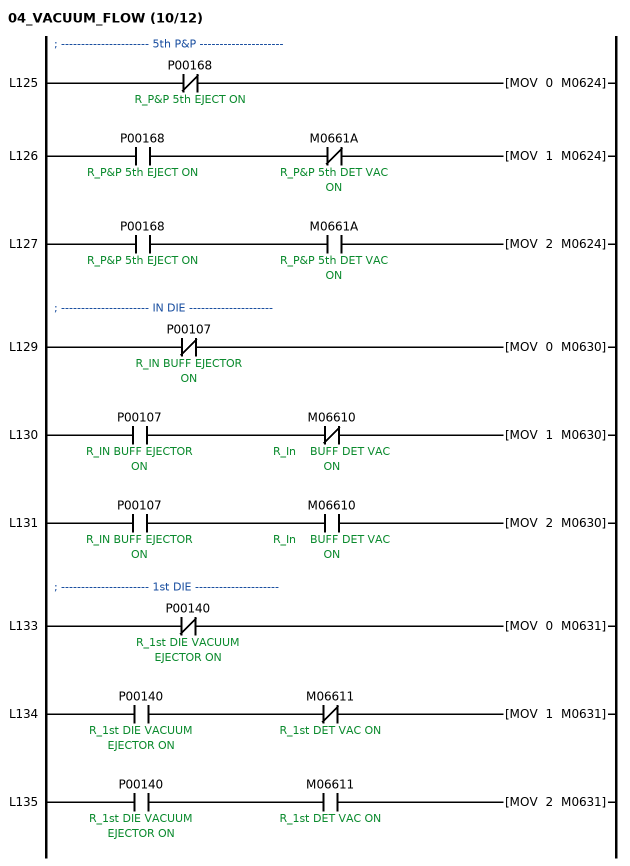
// ---------------------- 5th P&P ---------------------
; L125
LOAD NOT  P00168	// R_P&P 5th EJECT ON
MOV       0 M0624
; L126
LOAD      P00168	// R_P&P 5th EJECT ON
AND NOT   M0661A	// R_P&P 5th DET VAC ON
MOV       1 M0624
; L127
LOAD      P00168	// R_P&P 5th EJECT ON
AND       M0661A	// R_P&P 5th DET VAC ON
MOV       2 M0624
// ---------------------- IN DIE ---------------------
; L129
LOAD NOT  P00107	// R_IN BUFF EJECTOR ON
MOV       0 M0630
; L130
LOAD      P00107	// R_IN BUFF EJECTOR ON
AND NOT   M06610	// R_In    BUFF DET VAC ON
MOV       1 M0630
; L131
LOAD      P00107	// R_IN BUFF EJECTOR ON
AND       M06610	// R_In    BUFF DET VAC ON
MOV       2 M0630
// ---------------------- 1st DIE ---------------------
; L133
LOAD NOT  P00140	// R_1st DIE VACUUM EJECTOR ON
MOV       0 M0631
; L134
LOAD      P00140	// R_1st DIE VACUUM EJECTOR ON
AND NOT   M06611	// R_1st DET VAC ON
MOV       1 M0631
; L135
LOAD      P00140	// R_1st DIE VACUUM EJECTOR ON
AND       M06611	// R_1st DET VAC ON
MOV       2 M0631

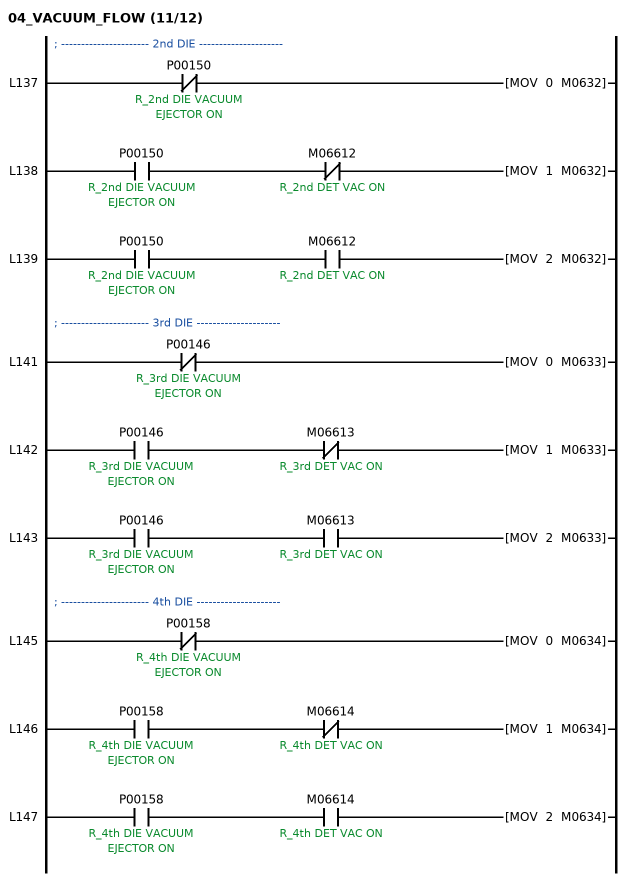
// ---------------------- 2nd DIE ---------------------
; L137
LOAD NOT  P00150	// R_2nd DIE VACUUM EJECTOR ON
MOV       0 M0632
; L138
LOAD      P00150	// R_2nd DIE VACUUM EJECTOR ON
AND NOT   M06612	// R_2nd DET VAC ON
MOV       1 M0632
; L139
LOAD      P00150	// R_2nd DIE VACUUM EJECTOR ON
AND       M06612	// R_2nd DET VAC ON
MOV       2 M0632
// ---------------------- 3rd DIE ---------------------
; L141
LOAD NOT  P00146	// R_3rd DIE VACUUM EJECTOR ON
MOV       0 M0633
; L142
LOAD      P00146	// R_3rd DIE VACUUM EJECTOR ON
AND NOT   M06613	// R_3rd DET VAC ON
MOV       1 M0633
; L143
LOAD      P00146	// R_3rd DIE VACUUM EJECTOR ON
AND       M06613	// R_3rd DET VAC ON
MOV       2 M0633
// ---------------------- 4th DIE ---------------------
; L145
LOAD NOT  P00158	// R_4th DIE VACUUM EJECTOR ON
MOV       0 M0634
; L146
LOAD      P00158	// R_4th DIE VACUUM EJECTOR ON
AND NOT   M06614	// R_4th DET VAC ON
MOV       1 M0634
; L147
LOAD      P00158	// R_4th DIE VACUUM EJECTOR ON
AND       M06614	// R_4th DET VAC ON
MOV       2 M0634

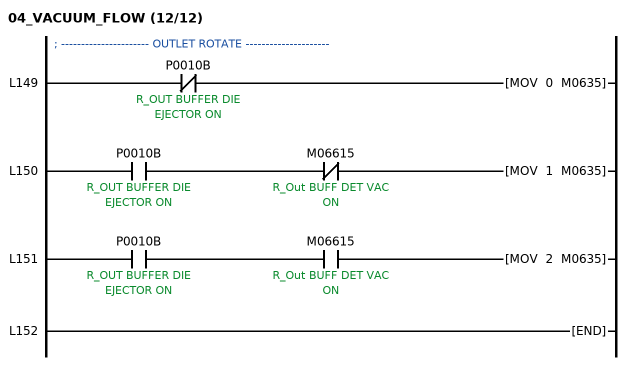
// ---------------------- OUTLET ROTATE ---------------------
; L149
LOAD NOT  P0010B	// R_OUT BUFFER DIE EJECTOR ON
MOV       0 M0635
; L150
LOAD      P0010B	// R_OUT BUFFER DIE EJECTOR ON
AND NOT   M06615	// R_Out BUFF DET VAC ON
MOV       1 M0635
; L151
LOAD      P0010B	// R_OUT BUFFER DIE EJECTOR ON
AND       M06615	// R_Out BUFF DET VAC ON
MOV       2 M0635
; L152
END

PROGRAM 05_TACKTIME_LOG (task: ½ºÄµ ÇÁ·Î±×·¥)

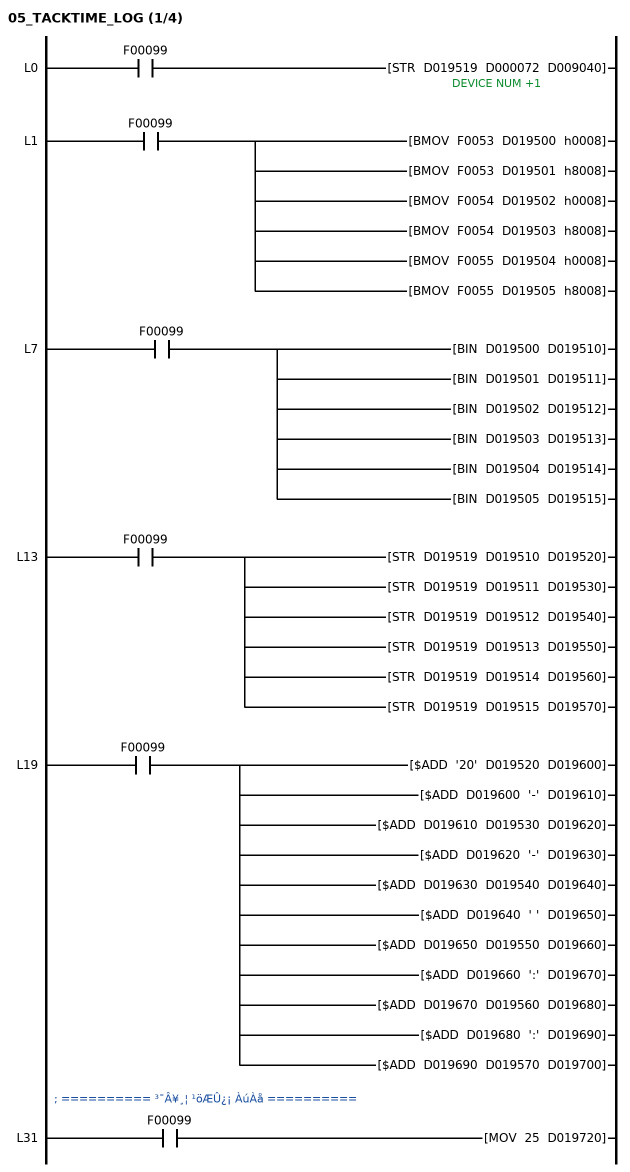
; L0
LOAD      F00099
STR       D019519 D000072 D009040	// DEVICE NUM +1
; L1
LOAD      F00099
BMOV      F0053 D019500 h0008
BMOV      F0053 D019501 h8008
BMOV      F0054 D019502 h0008
BMOV      F0054 D019503 h8008
BMOV      F0055 D019504 h0008
BMOV      F0055 D019505 h8008
; L7
LOAD      F00099
BIN       D019500 D019510
BIN       D019501 D019511
BIN       D019502 D019512
BIN       D019503 D019513
BIN       D019504 D019514
BIN       D019505 D019515
; L13
LOAD      F00099
STR       D019519 D019510 D019520
STR       D019519 D019511 D019530
STR       D019519 D019512 D019540
STR       D019519 D019513 D019550
STR       D019519 D019514 D019560
STR       D019519 D019515 D019570
; L19
LOAD      F00099
$ADD      '20' D019520 D019600
$ADD      D019600 '-' D019610
$ADD      D019610 D019530 D019620
$ADD      D019620 '-' D019630
$ADD      D019630 D019540 D019640
$ADD      D019640 ' ' D019650
$ADD      D019650 D019550 D019660
$ADD      D019660 ':' D019670
$ADD      D019670 D019560 D019680
$ADD      D019680 ':' D019690
$ADD      D019690 D019570 D019700
// ========== ³¯Â¥¸¦ ¹öÆÛ¿¡ ÀúÀå ==========
; L31
LOAD      F00099
MOV       25 D019720

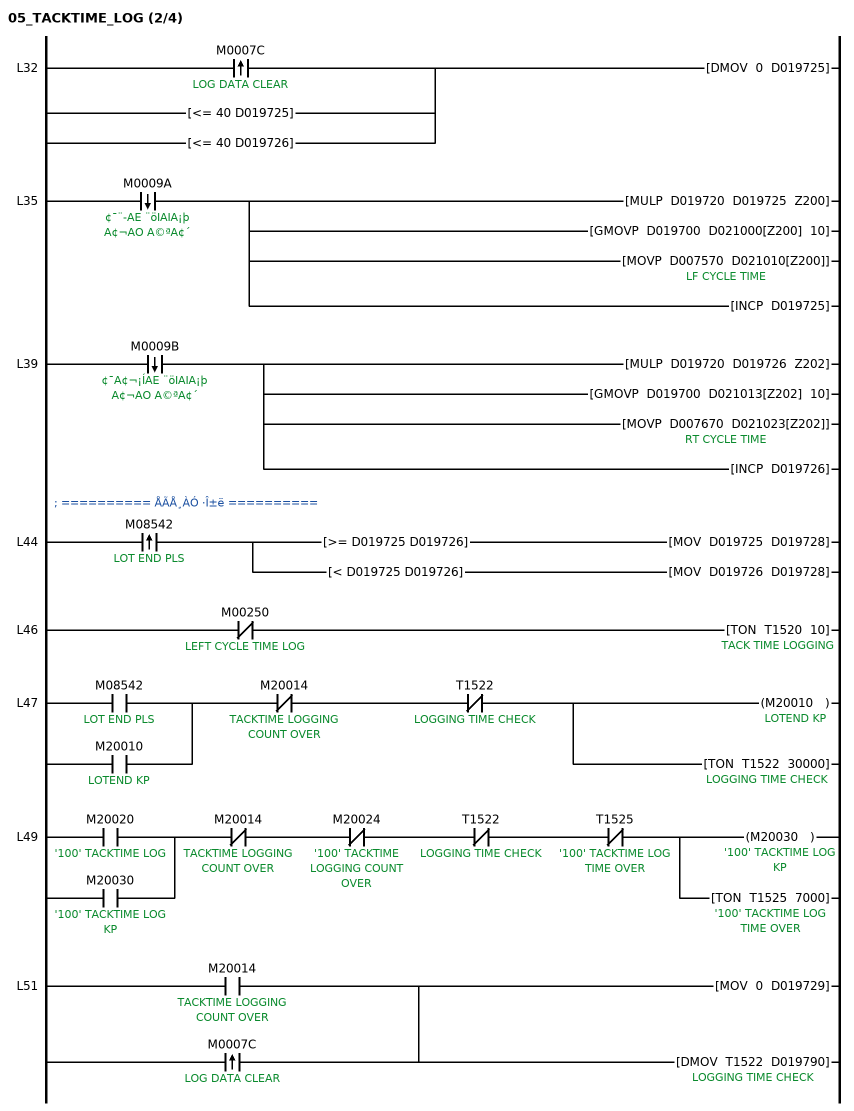
; L32
LOADP     M0007C	// LOG DATA CLEAR
OR<=      40 D019725
OR<=      40 D019726
DMOV      0 D019725
; L35
LOADN     M0009A	// ¢¯¨­AE ¨öIAIA¡þ A¢¬AO A©ªA¢´
MULP      D019720 D019725 Z200
GMOVP     D019700 D021000[Z200] 10
MOVP      D007570 D021010[Z200]	// LF CYCLE TIME
INCP      D019725
; L39
LOADN     M0009B	// ¢¯A¢¬¡ÍAE ¨öIAIA¡þ A¢¬AO A©ªA¢´
MULP      D019720 D019726 Z202
GMOVP     D019700 D021013[Z202] 10
MOVP      D007670 D021023[Z202]	// RT CYCLE TIME
INCP      D019726
// ========== ÅÃÅ¸ÀÓ ·Î±ë ==========
; L44
LOADP     M08542	// LOT END PLS
MPUSH
AND>=     D019725 D019726
MOV       D019725 D019728
MPOP
AND<      D019725 D019726
MOV       D019726 D019728
; L46
LOAD NOT  M00250	// LEFT CYCLE TIME LOG
TON       T1520 10	// TACK TIME LOGGING
; L47
LOAD      M08542	// LOT END PLS
OR        M20010	// LOTEND KP
AND NOT   M20014	// TACKTIME LOGGING COUNT OVER
AND NOT   T1522	// LOGGING TIME CHECK
OUT       M20010	// LOTEND KP
TON       T1522 30000	// LOGGING TIME CHECK
; L49
LOAD      M20020	// '100' TACKTIME LOG 
OR        M20030	// '100' TACKTIME LOG KP
AND NOT   M20014	// TACKTIME LOGGING COUNT OVER
AND NOT   M20024	// '100' TACKTIME LOGGING COUNT OVER
AND NOT   T1522	// LOGGING TIME CHECK
AND NOT   T1525	// '100' TACKTIME LOG TIME OVER
OUT       M20030	// '100' TACKTIME LOG KP
TON       T1525 7000	// '100' TACKTIME LOG TIME OVER
; L51
LOAD      M20014	// TACKTIME LOGGING COUNT OVER
ORP       M0007C	// LOG DATA CLEAR
MOV       0 D019729
DMOV      T1522 D019790	// LOGGING TIME CHECK

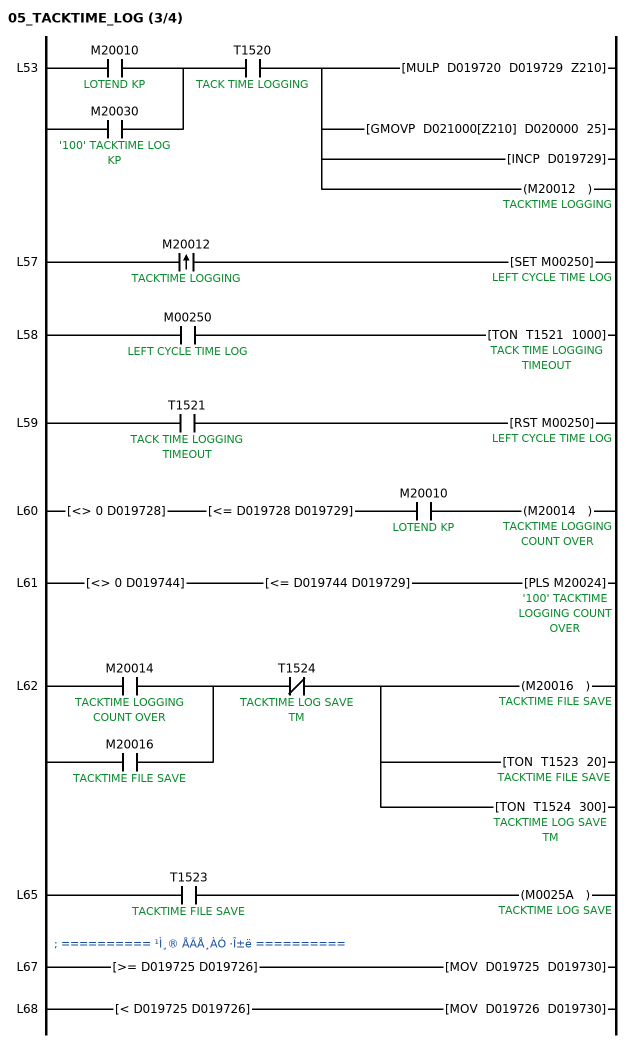
; L53
LOAD      M20010	// LOTEND KP
OR        M20030	// '100' TACKTIME LOG KP
AND       T1520	// TACK TIME LOGGING
MULP      D019720 D019729 Z210
GMOVP     D021000[Z210] D020000 25
INCP      D019729
OUT       M20012	// TACKTIME LOGGING
; L57
LOADP     M20012	// TACKTIME LOGGING
SET       M00250	// LEFT CYCLE TIME LOG
; L58
LOAD      M00250	// LEFT CYCLE TIME LOG
TON       T1521 1000	// TACK TIME LOGGING TIMEOUT
; L59
LOAD      T1521	// TACK TIME LOGGING TIMEOUT
RST       M00250	// LEFT CYCLE TIME LOG
; L60
LOAD<>    0 D019728
AND<=     D019728 D019729
AND       M20010	// LOTEND KP
OUT       M20014	// TACKTIME LOGGING COUNT OVER
; L61
LOAD<>    0 D019744
AND<=     D019744 D019729
OUTP      M20024	// '100' TACKTIME LOGGING COUNT OVER
; L62
LOAD      M20014	// TACKTIME LOGGING COUNT OVER
OR        M20016	// TACKTIME FILE SAVE
AND NOT   T1524	// TACKTIME LOG SAVE TM
OUT       M20016	// TACKTIME FILE SAVE
TON       T1523 20	// TACKTIME FILE SAVE
TON       T1524 300	// TACKTIME LOG SAVE TM
; L65
LOAD      T1523	// TACKTIME FILE SAVE
OUT       M0025A	// TACKTIME LOG SAVE
// ========== ¹Ì¸® ÅÃÅ¸ÀÓ ·Î±ë ==========
; L67
LOAD>=    D019725 D019726
MOV       D019725 D019730
; L68
LOAD<     D019725 D019726
MOV       D019726 D019730

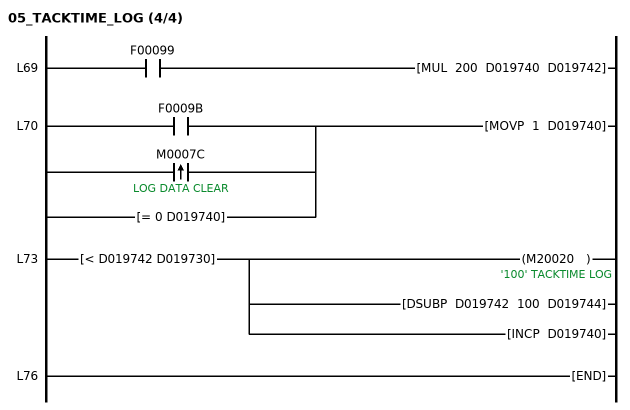
; L69
LOAD      F00099
MUL       200 D019740 D019742
; L70
LOAD      F0009B
ORP       M0007C	// LOG DATA CLEAR
OR=       0 D019740
MOVP      1 D019740
; L73
LOAD<     D019742 D019730
OUT       M20020	// '100' TACKTIME LOG 
DSUBP     D019742 100 D019744
INCP      D019740
; L76
END

PROGRAM 06_IO (task: ½ºÄµ ÇÁ·Î±×·¥)

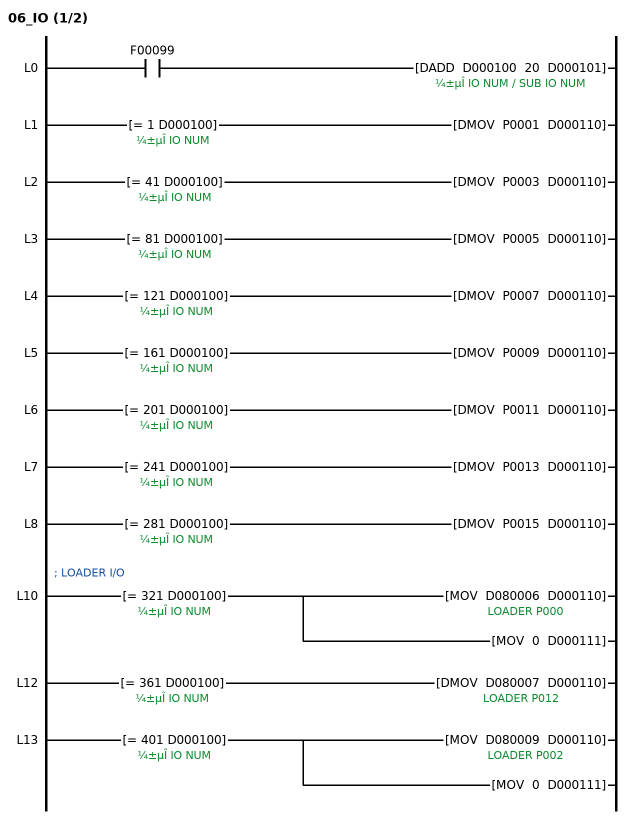
; L0
LOAD      F00099
DADD      D000100 20 D000101	// ¼±µÎ IO NUM / SUB IO NUM
; L1
LOAD=     1 D000100	// ¼±µÎ IO NUM
DMOV      P0001 D000110
; L2
LOAD=     41 D000100	// ¼±µÎ IO NUM
DMOV      P0003 D000110
; L3
LOAD=     81 D000100	// ¼±µÎ IO NUM
DMOV      P0005 D000110
; L4
LOAD=     121 D000100	// ¼±µÎ IO NUM
DMOV      P0007 D000110
; L5
LOAD=     161 D000100	// ¼±µÎ IO NUM
DMOV      P0009 D000110
; L6
LOAD=     201 D000100	// ¼±µÎ IO NUM
DMOV      P0011 D000110
; L7
LOAD=     241 D000100	// ¼±µÎ IO NUM
DMOV      P0013 D000110
; L8
LOAD=     281 D000100	// ¼±µÎ IO NUM
DMOV      P0015 D000110
// LOADER I/O
; L10
LOAD=     321 D000100	// ¼±µÎ IO NUM
MOV       D080006 D000110	// LOADER P000
MOV       0 D000111
; L12
LOAD=     361 D000100	// ¼±µÎ IO NUM
DMOV      D080007 D000110	// LOADER P012
; L13
LOAD=     401 D000100	// ¼±µÎ IO NUM
MOV       D080009 D000110	// LOADER P002
MOV       0 D000111

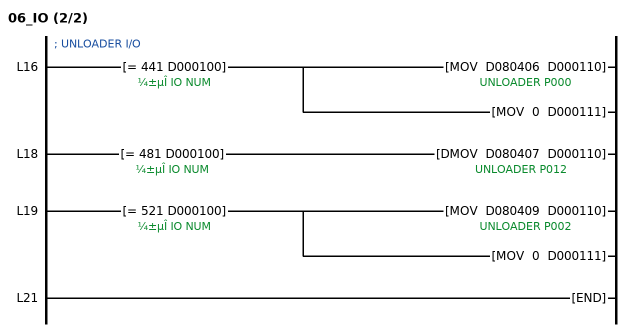
// UNLOADER I/O
; L16
LOAD=     441 D000100	// ¼±µÎ IO NUM
MOV       D080406 D000110	// UNLOADER P000
MOV       0 D000111
; L18
LOAD=     481 D000100	// ¼±µÎ IO NUM
DMOV      D080407 D000110	// UNLOADER P012
; L19
LOAD=     521 D000100	// ¼±µÎ IO NUM
MOV       D080409 D000110	// UNLOADER P002
MOV       0 D000111
; L21
END

PROGRAM 07_VACUUM (task: ½ºÄµ ÇÁ·Î±×·¥)

